// TIA Portal V20 export
// export: Created 2025-12-01T14:56:43.4302356Z, ExportSetting None, DisplayName Totally Integrated Automation Portal, DisplayVersion V20 Update 3, DisplayName TIA Portal Openness, DisplayVersion V20 Update 3, DisplayName TIA Portal Version Control Interface, DisplayVersion V20 Update 3, DisplayName STEP 7 Professional, DisplayVersion V20 Update 3, DisplayName STEP 7 Safety, DisplayVersion V20 Update 2, DisplayName WinCC Basic/Comfort/Advanced, DisplayVersion V20 Update 3, DisplayName WinCC Professional, DisplayVersion V20 Update 3, DisplayName WinCC Unified, DisplayVersion V20 Update 3
FUNCTION_BLOCK "FB243_M_STV_Carga_E1_S3_Doble"   // FB243, LAD
TITLE = Control del Ramal de Salidas
{ S7_Optimized_Access := 'FALSE' }
AUTHOR : VTD
NAME : 20160509
VERSION : 3.5
// stored: AutoNumber false, SetENOAutomatically false
   VAR_INPUT
      Mesa : UInt;   // Mesa de la FB
      Error_Tx : Bool;   // Error en el Tx
      EnTension : Bool;   // Existe Tension en la Mesa
      Termico_Tx : Bool;   // Proteccion del Tx
      pHsMx_1 : Bool;   // pHs de la Mesa
      pHsMx_2 : Bool;   // pHs de la Mesa
      pHsMx_PR1 : Bool;   // pHs de Protrusion de la Mesa. Nota: No existe >> ON
      pHsMx_PR3 : Bool;   // pHs de Protrusion de la Mesa. Nota: No existe >> ON
      Avance_Tx : Bool;   // Avance del Tx
      LoadArrival : Bool;   // Load Arrival >>> VTD
      LoadComplete : Bool;   // LoadComplete >>> VTD
      MAnt_DescargaAct : Bool;   // E1 >> Mesa Anterior DescargaAct
      AVTF_MAnt_Mx : Bool;   // E1 >> Mesa Anterior AVTF
      P_Mens_MAnt_Mx : Bool;   // E1 >> Mesa Anterior P_Mens
      MAnt_CargaLarga : Bool;   // E1 >> Mesa Anterior Carga Larga
      Mx_VelocidadLenta_In : Bool;   // Forzar a Velociada Lenta
      F_EnvMens_Mx : Bool;   // Fin de Envio de Mensaje
      OrdSal_S00 : Bool;   // Orden de Salida hacia el VTD
      V_CNT_pHsMx : Int := 1000;   // Valor de Presencia
      V_CNT_pHsMx_FTF : Int := 200;   // Valor para activar FTF. Nota: < = V_CNT_pHsMx.
      V_CNTSeg_pHsMx : Int := 2000;   // Valor de Seguriadad para Presencia
      V_CNT_PasoLenta : Int := 2000;   // Valor de Paso a Lenta
      V_CNT_ApHsMx : Int := 200;   // Valor de Ausencia
      V_CNTSeg_ApHsMx : Int := 2000;   // Valor de Seguriadad para Ausencia
      V_TOut_Tx_Mx : Int := 15000;   // TimeOut de Entrada por E1
      V_TOut_Interlock : Int := 5000;   // TimeOut de Fin del Interlock con el VTD
      V_TMP_Protrusion : Int := 200;   // TMP de Protrusion
      V_CNT_PerdidapHs : Int := 1000;   // CNT de Perdida de pHs
   END_VAR
   VAR_OUTPUT
      P_EnvMens_PMx : Bool;   // Permiso de Enviar Mensaje de Presencia
      P_EnvMens_AMx : Bool;   // Permiso de Enviar Mensaje de Ausencia
      P_RecepOK_Mx : Bool;   // Recepcion OK
      PTF_MAnt_Mx : Bool;   // E1 >> Mesa Anterior PTF
      FTF_MAnt_Mx : Bool;   // E1 >> Mesa Anterior FTF
   END_VAR
   VAR
      Anular_prE1 : Bool;   // ???
      Anular_prS3 : Bool;   // ???
      Mx_ET00 : Bool;
      Mx_ET01 : Bool;
      Mx_ET02 : Bool;
      Mx_ET06 : Bool;
      Mx_ET07 : Bool;
      Mx_ET08 : Bool;
      Mx_ET09 : Bool;
      Mx_ET10 : Bool;
      Mx_ET10Doble : Bool;
      Mx_ET11 : Bool;
      Mx_ET12 : Bool;
      Mx_ET110 : Bool;
      Mx_ET111 : Bool;
      Mx_ET50 : Bool;
      Mx_ET51 : Bool;
      Mx_ET52 : Bool;
      Mx_ET150 : Bool;
      Mx_ET151 : Bool;
      Mx_ET152 : Bool;
      MemoriaCargaDoble : Bool;   // Interna >>> Memoria Carga Doble
      ProtocoloIniciado : Bool;   // Iniciado el Envio del Mensaje de Presencia
      CNT_pHsMx_FTF_OK : Bool;   // Enviar ya FTF
      STAT_EnvMens_PMx : Bool;   // Interna >> Envio del Mensaje de Presencia
      STAT_EnvMens_AMx : Bool;   // Interna >> Envio de Mensaje de Ausencia
      STAT_FTF_MAnt_Mx : Bool;   // Interna >> FTF de MAnt >> Mx
      CNT_pHsMx { S7_SetPoint := 'True'} : "FB910_CNT_UHS";   // CNT de la Presencia
      CNTSeg_pHsMx { S7_SetPoint := 'True'} : "FB910_CNT_UHS";   // CNT de Seguridad de la Presencia
      CNT_ApHsMx { S7_SetPoint := 'True'} : "FB910_CNT_UHS";   // CNT de la Ausencia
      CNTSeg_ApHsMx { S7_SetPoint := 'True'} : "FB910_CNT_UHS";   // CNT de Seguridad de la Ausencia
      TMP_EnTension { S7_SetPoint := 'True'} : "FB910_CNT_UHS";
      TOut_Av_Mx { S7_SetPoint := 'True'} : "FB910_CNT_UHS";   // Time Out de Entrada de E1
      TOut_Interlock { S7_SetPoint := 'True'} : "FB910_CNT_UHS";   // Time Out de Fin de Interlock con el VTD
      TMP_Protrusion { S7_SetPoint := 'True'} : "FB910_CNT_UHS";   // TMP de la Protrusion
      Interlock_manual { S7_SetPoint := 'True'} : "UDT_Interlock_manual_STV";
      CNT_PerdidapHs { S7_SetPoint := 'True'} : "FB910_CNT_UHS";   // CNT de Perdida de pHs
   END_VAR
   VAR_TEMP
      EstadoZona : "EstadoZona";   // Estado de Zona de la Mesa
      EstadoVI : "EstadosMesa";   // Estado del Vehiculo Inteliguente de la Mesa
      ConfigFB : "UDT_ConfigFB";   // Configuracion de la FB de la Mesa
      Interlock : "UDT_Interlock_STV";
      V_Protrusion : Int;
      retval : Int;
      cero : USInt;
      Aux_ET00 : Bool;
   END_VAR
BEGIN

REGION Network 1: INICIALIZAR - Recoger las Variables de Estado de la Mesa
   // Se recoge - Estado_CBx
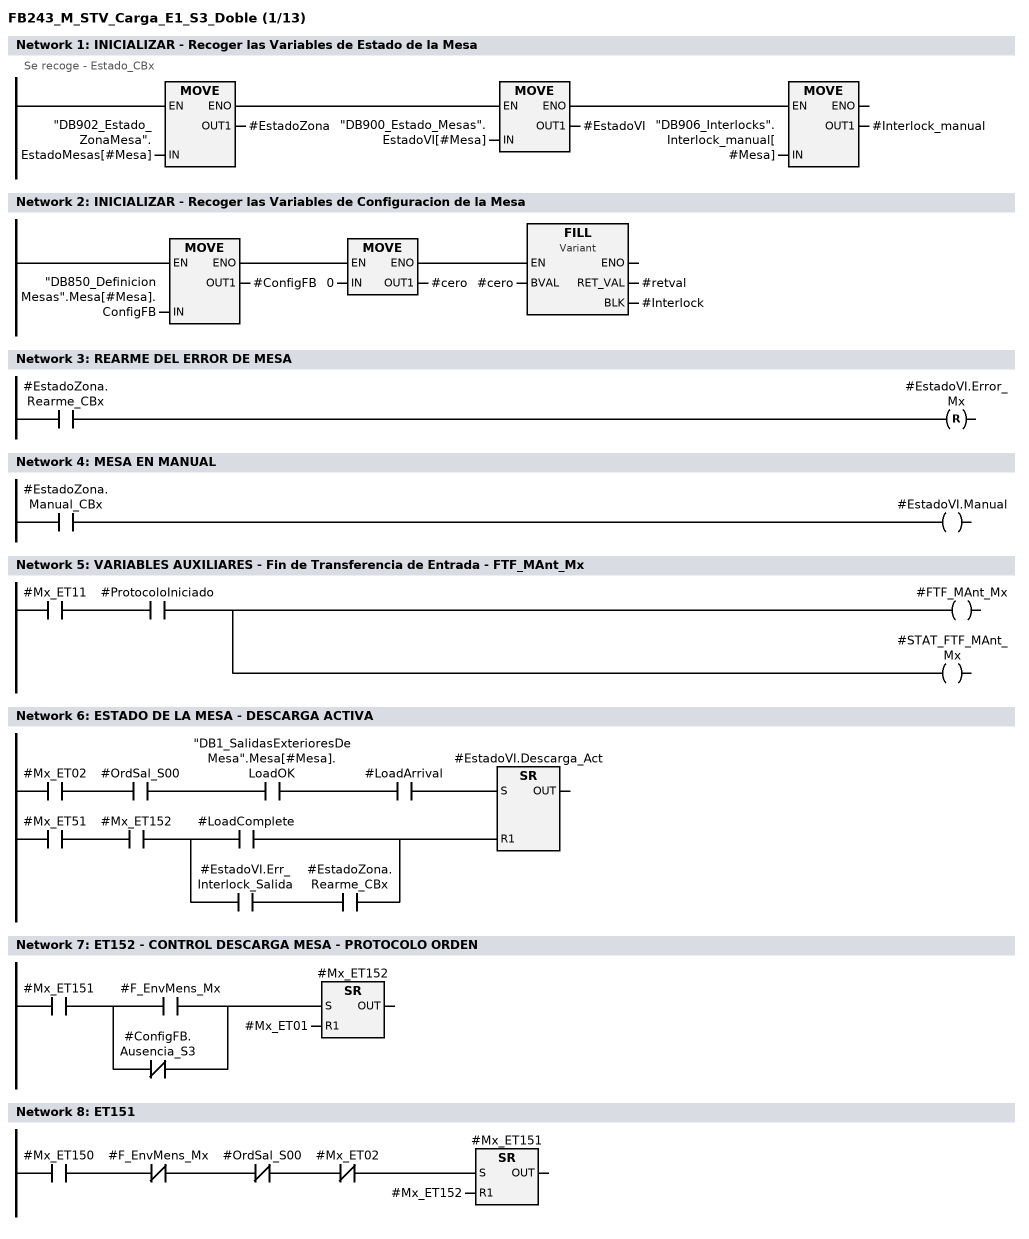
   RUNG wire#powerrail
      Move(in := "DB902_Estado_ZonaMesa".EstadoMesas[#Mesa], out1 => #EstadoZona)
      Move(in := "DB900_Estado_Mesas".EstadoVI[#Mesa], out1 => #EstadoVI)
      Move(in := "DB906_Interlocks".Interlock_manual[#Mesa], out1 => #Interlock_manual)
   END_RUNG
   // the same network as SCL:
   #EstadoZona := "DB902_Estado_ZonaMesa".EstadoMesas[#Mesa];
   #EstadoVI := "DB900_Estado_Mesas".EstadoVI[#Mesa];
   #Interlock_manual := "DB906_Interlocks".Interlock_manual[#Mesa];
END_REGION

REGION Network 2: INICIALIZAR - Recoger las Variables de Configuracion de la Mesa
   RUNG wire#powerrail
      Move(in := "DB850_DefinicionMesas".Mesa[#Mesa].ConfigFB, out1 => #ConfigFB)
      Move(in := 0, out1 => #cero)
      { S7_Templates := "ptr_type := Variant" } FILL(BVAL := #cero, RET_VAL => #retval, BLK => #Interlock)
   END_RUNG
   // the same network as SCL:
   #ConfigFB := "DB850_DefinicionMesas".Mesa[#Mesa].ConfigFB;
   #cero := 0;
   #retval := FILL(BVAL := #cero, BLK => #Interlock);
END_REGION

REGION Network 3: REARME DEL ERROR DE MESA
   RUNG wire#powerrail
      Contact( #EstadoZona.Rearme_CBx )
      R_Coil( #EstadoVI.Error_Mx )
   END_RUNG
   // the same network as SCL:
   IF #EstadoZona.Rearme_CBx THEN #EstadoVI.Error_Mx := FALSE; END_IF;
END_REGION

REGION Network 4: MESA EN MANUAL
   RUNG wire#powerrail
      Contact( #EstadoZona.Manual_CBx )
      Coil( #EstadoVI.Manual )
   END_RUNG
   // the same network as SCL:
   #EstadoVI.Manual := #EstadoZona.Manual_CBx;
END_REGION

REGION Network 5: VARIABLES AUXILIARES - Fin de Transferencia de Entrada - FTF_MAnt_Mx
   RUNG wire#powerrail
      Contact( #Mx_ET11 )
      Contact( #ProtocoloIniciado )
      wire#w1
      Coil( #FTF_MAnt_Mx )
   END_RUNG
   RUNG wire#w1
      Coil( #STAT_FTF_MAnt_Mx )
   END_RUNG
   // the same network as SCL:
   #FTF_MAnt_Mx := #Mx_ET11 AND #ProtocoloIniciado;
   #STAT_FTF_MAnt_Mx := #FTF_MAnt_Mx;
END_REGION

REGION Network 6: ESTADO DE LA MESA - DESCARGA ACTIVA
   RUNG wire#powerrail
      Contact( #Mx_ET02 )
      Contact( #OrdSal_S00 )
      Contact( "DB1_SalidasExterioresDeMesa".Mesa[#Mesa].LoadOK )
      Contact( #LoadArrival )
      S_SR(operand := #EstadoVI.Descarga_Act, r1 := wire#w2)
   END_RUNG
   RUNG wire#powerrail
      Contact( #Mx_ET51 )
      Contact( #Mx_ET152 )
      wire#w1
      Contact( #LoadComplete )
   END_RUNG wire#w2
   RUNG wire#w1
      Contact( #EstadoVI.Err_Interlock_Salida )
      Contact( #EstadoZona.Rearme_CBx )
   END_RUNG wire#w2
   // the same network as SCL:
   IF #Mx_ET02 AND #OrdSal_S00 AND "DB1_SalidasExterioresDeMesa".Mesa[#Mesa].LoadOK AND #LoadArrival THEN
       #EstadoVI.Descarga_Act := TRUE;   // SR flip-flop
   END_IF;
   IF #Mx_ET51 AND #Mx_ET152 AND (#LoadComplete OR (#EstadoVI.Err_Interlock_Salida AND #EstadoZona.Rearme_CBx)) THEN
       #EstadoVI.Descarga_Act := FALSE;
   END_IF;
END_REGION

REGION Network 7: ET152 - CONTROL DESCARGA MESA - PROTOCOLO ORDEN
   RUNG wire#powerrail
      Contact( #Mx_ET151 )
      wire#w1
      Contact( #F_EnvMens_Mx )
      wire#w2
      S_SR(operand := #Mx_ET152, r1 := #Mx_ET01)
   END_RUNG
   RUNG wire#w1
      I_Contact( #ConfigFB.Ausencia_S3 )
   END_RUNG wire#w2
   // the same network as SCL:
   IF #Mx_ET151 AND (#F_EnvMens_Mx OR NOT #ConfigFB.Ausencia_S3) THEN
       #Mx_ET152 := TRUE;   // SR flip-flop
   END_IF;
   IF #Mx_ET01 THEN #Mx_ET152 := FALSE; END_IF;
END_REGION

REGION Network 8: ET151
   RUNG wire#powerrail
      Contact( #Mx_ET150 )
      I_Contact( #F_EnvMens_Mx )
      I_Contact( #OrdSal_S00 )
      I_Contact( #Mx_ET02 )
      S_SR(operand := #Mx_ET151, r1 := #Mx_ET152)
   END_RUNG
   // the same network as SCL:
   IF #Mx_ET150 AND NOT #F_EnvMens_Mx AND NOT #OrdSal_S00 AND NOT #Mx_ET02 THEN
       #Mx_ET151 := TRUE;   // SR flip-flop
   END_IF;
   IF #Mx_ET152 THEN #Mx_ET151 := FALSE; END_IF;
END_REGION

REGION Network 9: ET150
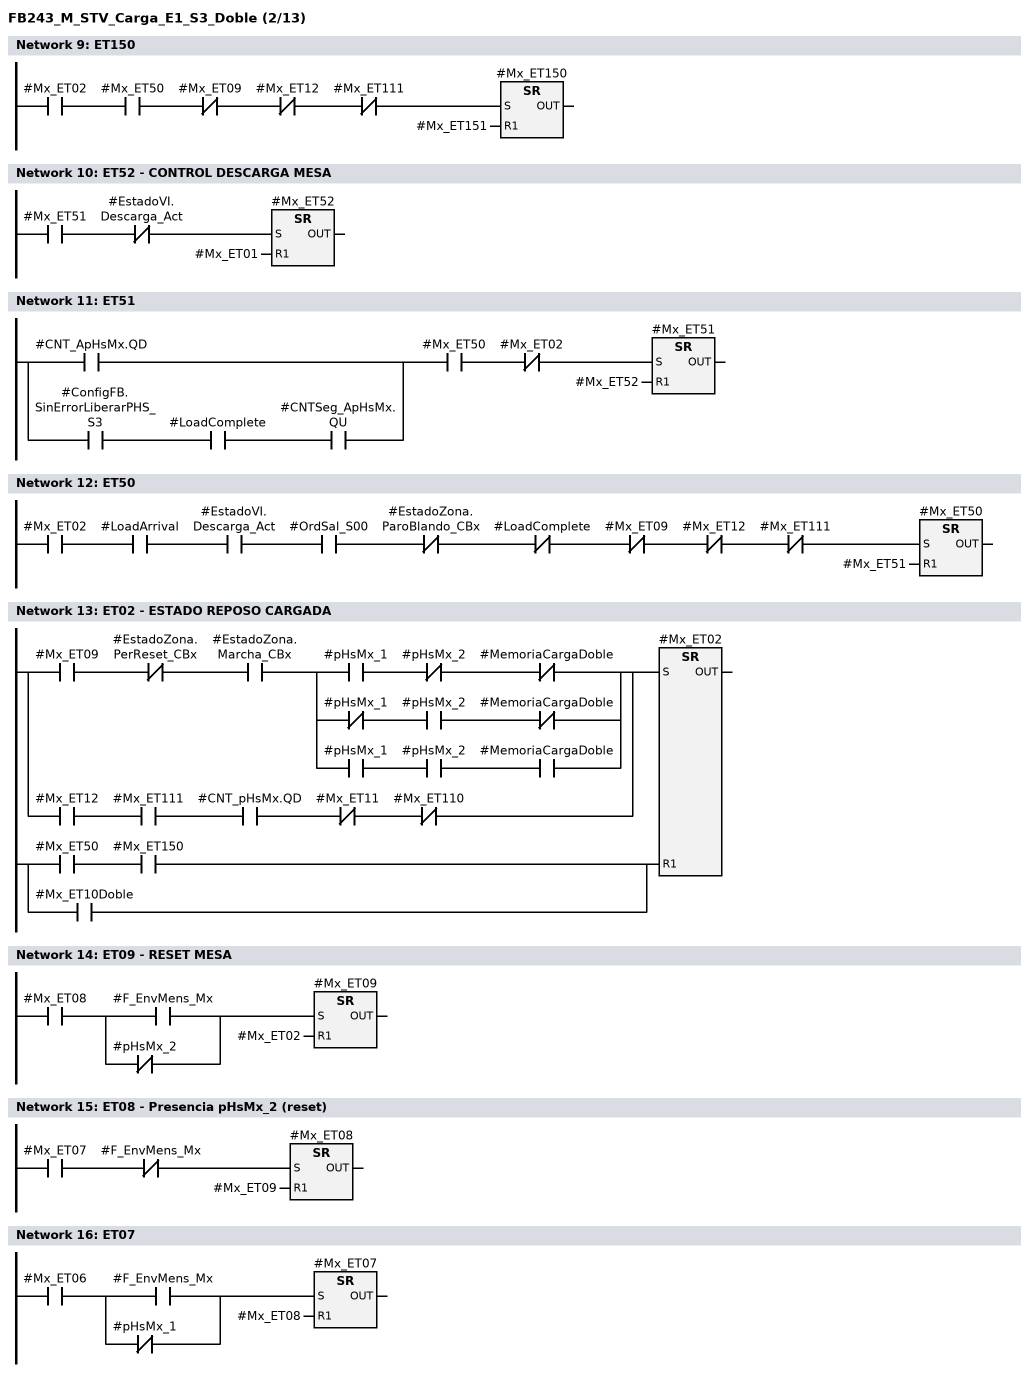
   RUNG wire#powerrail
      Contact( #Mx_ET02 )
      Contact( #Mx_ET50 )
      I_Contact( #Mx_ET09 )
      I_Contact( #Mx_ET12 )
      I_Contact( #Mx_ET111 )
      S_SR(operand := #Mx_ET150, r1 := #Mx_ET151)
   END_RUNG
   // the same network as SCL:
   IF #Mx_ET02 AND #Mx_ET50 AND NOT #Mx_ET09 AND NOT #Mx_ET12 AND NOT #Mx_ET111 THEN
       #Mx_ET150 := TRUE;   // SR flip-flop
   END_IF;
   IF #Mx_ET151 THEN #Mx_ET150 := FALSE; END_IF;
END_REGION

REGION Network 10: ET52 - CONTROL DESCARGA MESA
   RUNG wire#powerrail
      Contact( #Mx_ET51 )
      I_Contact( #EstadoVI.Descarga_Act )
      S_SR(operand := #Mx_ET52, r1 := #Mx_ET01)
   END_RUNG
   // the same network as SCL:
   IF #Mx_ET51 AND NOT #EstadoVI.Descarga_Act THEN
       #Mx_ET52 := TRUE;   // SR flip-flop
   END_IF;
   IF #Mx_ET01 THEN #Mx_ET52 := FALSE; END_IF;
END_REGION

REGION Network 11: ET51
   RUNG wire#powerrail
      Contact( #CNT_ApHsMx.QD )
      wire#w1
      Contact( #Mx_ET50 )
      I_Contact( #Mx_ET02 )
      S_SR(operand := #Mx_ET51, r1 := #Mx_ET52)
   END_RUNG
   RUNG wire#powerrail
      Contact( #ConfigFB.SinErrorLiberarPHS_S3 )
      Contact( #LoadComplete )
      Contact( #CNTSeg_ApHsMx.QU )
   END_RUNG wire#w1
   // the same network as SCL:
   IF (#CNT_ApHsMx.QD OR (#ConfigFB.SinErrorLiberarPHS_S3 AND #LoadComplete AND #CNTSeg_ApHsMx.QU)) AND #Mx_ET50 AND NOT #Mx_ET02 THEN
       #Mx_ET51 := TRUE;   // SR flip-flop
   END_IF;
   IF #Mx_ET52 THEN #Mx_ET51 := FALSE; END_IF;
END_REGION

REGION Network 12: ET50
   RUNG wire#powerrail
      Contact( #Mx_ET02 )
      Contact( #LoadArrival )
      Contact( #EstadoVI.Descarga_Act )
      Contact( #OrdSal_S00 )
      I_Contact( #EstadoZona.ParoBlando_CBx )
      I_Contact( #LoadComplete )
      I_Contact( #Mx_ET09 )
      I_Contact( #Mx_ET12 )
      I_Contact( #Mx_ET111 )
      S_SR(operand := #Mx_ET50, r1 := #Mx_ET51)
   END_RUNG
   // the same network as SCL:
   IF #Mx_ET02 AND #LoadArrival AND #EstadoVI.Descarga_Act AND #OrdSal_S00 AND NOT #EstadoZona.ParoBlando_CBx AND NOT #LoadComplete AND NOT #Mx_ET09 AND NOT #Mx_ET12 AND NOT #Mx_ET111 THEN
       #Mx_ET50 := TRUE;   // SR flip-flop
   END_IF;
   IF #Mx_ET51 THEN #Mx_ET50 := FALSE; END_IF;
END_REGION

REGION Network 13: ET02 - ESTADO REPOSO CARGADA
   RUNG wire#powerrail
      Contact( #Mx_ET09 )
      I_Contact( #EstadoZona.PerReset_CBx )
      Contact( #EstadoZona.Marcha_CBx )
      wire#w1
      Contact( #pHsMx_1 )
      I_Contact( #pHsMx_2 )
      I_Contact( #MemoriaCargaDoble )
      wire#w2
      S_SR(operand := #Mx_ET02, r1 := wire#w3)
   END_RUNG
   RUNG wire#w1
      I_Contact( #pHsMx_1 )
      Contact( #pHsMx_2 )
      I_Contact( #MemoriaCargaDoble )
   END_RUNG wire#w2
   RUNG wire#w1
      Contact( #pHsMx_1 )
      Contact( #pHsMx_2 )
      Contact( #MemoriaCargaDoble )
   END_RUNG wire#w2
   RUNG wire#powerrail
      Contact( #Mx_ET12 )
      Contact( #Mx_ET111 )
      Contact( #CNT_pHsMx.QD )
      I_Contact( #Mx_ET11 )
      I_Contact( #Mx_ET110 )
   END_RUNG wire#w2
   RUNG wire#powerrail
      Contact( #Mx_ET50 )
      Contact( #Mx_ET150 )
   END_RUNG wire#w3
   RUNG wire#powerrail
      Contact( #Mx_ET10Doble )
   END_RUNG wire#w3
   // the same network as SCL:
   IF (#Mx_ET09 AND NOT #EstadoZona.PerReset_CBx AND #EstadoZona.Marcha_CBx AND ((#pHsMx_1 AND NOT #pHsMx_2 AND NOT #MemoriaCargaDoble) OR (NOT #pHsMx_1 AND #pHsMx_2 AND NOT #MemoriaCargaDoble) OR (#pHsMx_1 AND #pHsMx_2 AND #MemoriaCargaDoble))) OR (#Mx_ET12 AND #Mx_ET111 AND #CNT_pHsMx.QD AND NOT #Mx_ET11 AND NOT #Mx_ET110) THEN
       #Mx_ET02 := TRUE;   // SR flip-flop
   END_IF;
   IF (#Mx_ET50 AND #Mx_ET150) OR #Mx_ET10Doble THEN #Mx_ET02 := FALSE; END_IF;
END_REGION

REGION Network 14: ET09 - RESET MESA
   RUNG wire#powerrail
      Contact( #Mx_ET08 )
      wire#w1
      Contact( #F_EnvMens_Mx )
      wire#w2
      S_SR(operand := #Mx_ET09, r1 := #Mx_ET02)
   END_RUNG
   RUNG wire#w1
      I_Contact( #pHsMx_2 )
   END_RUNG wire#w2
   // the same network as SCL:
   IF #Mx_ET08 AND (#F_EnvMens_Mx OR NOT #pHsMx_2) THEN
       #Mx_ET09 := TRUE;   // SR flip-flop
   END_IF;
   IF #Mx_ET02 THEN #Mx_ET09 := FALSE; END_IF;
END_REGION

REGION Network 15: ET08 - Presencia pHsMx_2 (reset)
   RUNG wire#powerrail
      Contact( #Mx_ET07 )
      I_Contact( #F_EnvMens_Mx )
      S_SR(operand := #Mx_ET08, r1 := #Mx_ET09)
   END_RUNG
   // the same network as SCL:
   IF #Mx_ET07 AND NOT #F_EnvMens_Mx THEN
       #Mx_ET08 := TRUE;   // SR flip-flop
   END_IF;
   IF #Mx_ET09 THEN #Mx_ET08 := FALSE; END_IF;
END_REGION

REGION Network 16: ET07
   RUNG wire#powerrail
      Contact( #Mx_ET06 )
      wire#w1
      Contact( #F_EnvMens_Mx )
      wire#w2
      S_SR(operand := #Mx_ET07, r1 := #Mx_ET08)
   END_RUNG
   RUNG wire#w1
      I_Contact( #pHsMx_1 )
   END_RUNG wire#w2
   // the same network as SCL:
   IF #Mx_ET06 AND (#F_EnvMens_Mx OR NOT #pHsMx_1) THEN
       #Mx_ET07 := TRUE;   // SR flip-flop
   END_IF;
   IF #Mx_ET08 THEN #Mx_ET07 := FALSE; END_IF;
END_REGION

REGION Network 17: ET06 - Presencia pHsMx_1 (reset)
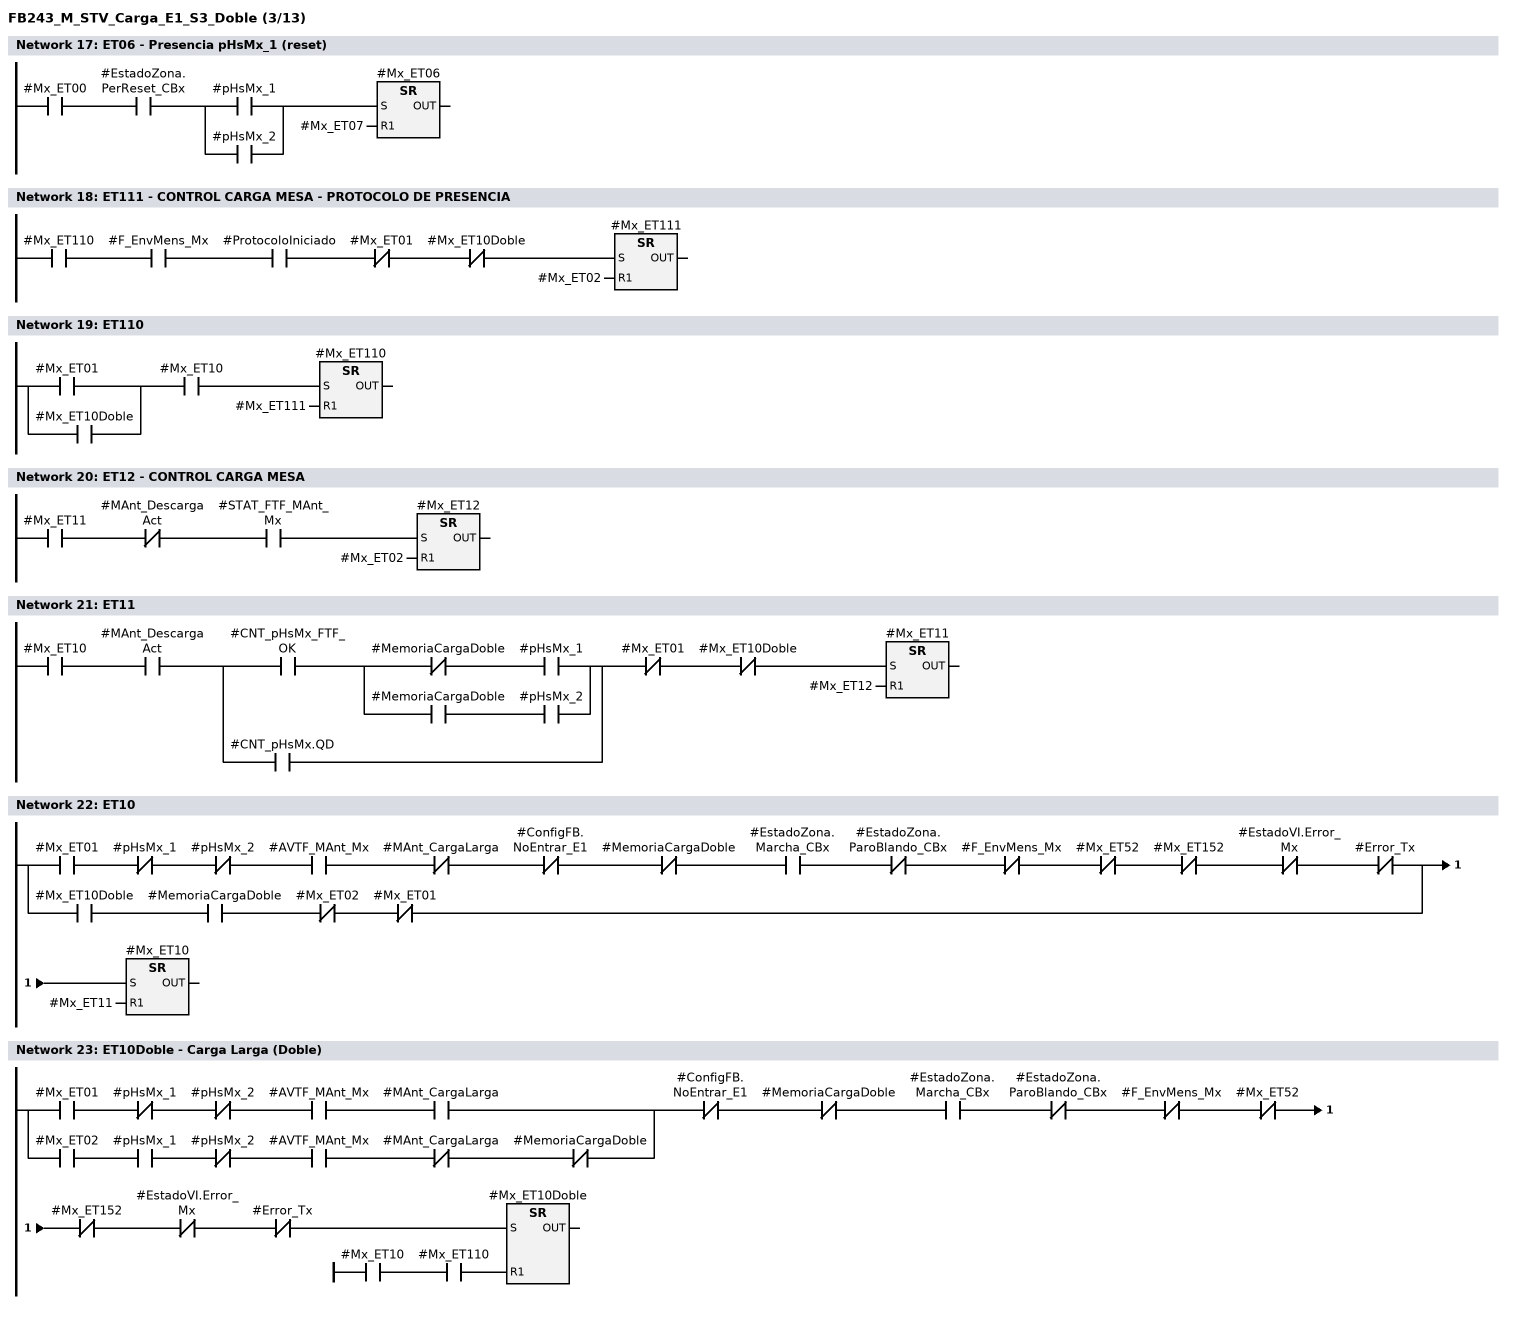
   RUNG wire#powerrail
      Contact( #Mx_ET00 )
      Contact( #EstadoZona.PerReset_CBx )
      wire#w1
      Contact( #pHsMx_1 )
      wire#w2
      S_SR(operand := #Mx_ET06, r1 := #Mx_ET07)
   END_RUNG
   RUNG wire#w1
      Contact( #pHsMx_2 )
   END_RUNG wire#w2
   // the same network as SCL:
   IF #Mx_ET00 AND #EstadoZona.PerReset_CBx AND (#pHsMx_1 OR #pHsMx_2) THEN
       #Mx_ET06 := TRUE;   // SR flip-flop
   END_IF;
   IF #Mx_ET07 THEN #Mx_ET06 := FALSE; END_IF;
END_REGION

REGION Network 18: ET111 - CONTROL CARGA MESA - PROTOCOLO DE PRESENCIA
   RUNG wire#powerrail
      Contact( #Mx_ET110 )
      Contact( #F_EnvMens_Mx )
      Contact( #ProtocoloIniciado )
      I_Contact( #Mx_ET01 )
      I_Contact( #Mx_ET10Doble )
      S_SR(operand := #Mx_ET111, r1 := #Mx_ET02)
   END_RUNG
   // the same network as SCL:
   IF #Mx_ET110 AND #F_EnvMens_Mx AND #ProtocoloIniciado AND NOT #Mx_ET01 AND NOT #Mx_ET10Doble THEN
       #Mx_ET111 := TRUE;   // SR flip-flop
   END_IF;
   IF #Mx_ET02 THEN #Mx_ET111 := FALSE; END_IF;
END_REGION

REGION Network 19: ET110
   RUNG wire#powerrail
      Contact( #Mx_ET01 )
      wire#w1
      Contact( #Mx_ET10 )
      S_SR(operand := #Mx_ET110, r1 := #Mx_ET111)
   END_RUNG
   RUNG wire#powerrail
      Contact( #Mx_ET10Doble )
   END_RUNG wire#w1
   // the same network as SCL:
   IF (#Mx_ET01 OR #Mx_ET10Doble) AND #Mx_ET10 THEN
       #Mx_ET110 := TRUE;   // SR flip-flop
   END_IF;
   IF #Mx_ET111 THEN #Mx_ET110 := FALSE; END_IF;
END_REGION

REGION Network 20: ET12 - CONTROL CARGA MESA
   RUNG wire#powerrail
      Contact( #Mx_ET11 )
      I_Contact( #MAnt_DescargaAct )
      Contact( #STAT_FTF_MAnt_Mx )
      S_SR(operand := #Mx_ET12, r1 := #Mx_ET02)
   END_RUNG
   // the same network as SCL:
   IF #Mx_ET11 AND NOT #MAnt_DescargaAct AND #STAT_FTF_MAnt_Mx THEN
       #Mx_ET12 := TRUE;   // SR flip-flop
   END_IF;
   IF #Mx_ET02 THEN #Mx_ET12 := FALSE; END_IF;
END_REGION

REGION Network 21: ET11
   RUNG wire#powerrail
      Contact( #Mx_ET10 )
      Contact( #MAnt_DescargaAct )
      wire#w1
      Contact( #CNT_pHsMx_FTF_OK )
      wire#w2
      I_Contact( #MemoriaCargaDoble )
      Contact( #pHsMx_1 )
      wire#w3
      I_Contact( #Mx_ET01 )
      I_Contact( #Mx_ET10Doble )
      S_SR(operand := #Mx_ET11, r1 := #Mx_ET12)
   END_RUNG
   RUNG wire#w2
      Contact( #MemoriaCargaDoble )
      Contact( #pHsMx_2 )
   END_RUNG wire#w3
   RUNG wire#w1
      Contact( #CNT_pHsMx.QD )
   END_RUNG wire#w3
   // the same network as SCL:
   IF #Mx_ET10 AND #MAnt_DescargaAct AND ((#CNT_pHsMx_FTF_OK AND ((NOT #MemoriaCargaDoble AND #pHsMx_1) OR (#MemoriaCargaDoble AND #pHsMx_2))) OR #CNT_pHsMx.QD) AND NOT #Mx_ET01 AND NOT #Mx_ET10Doble THEN
       #Mx_ET11 := TRUE;   // SR flip-flop
   END_IF;
   IF #Mx_ET12 THEN #Mx_ET11 := FALSE; END_IF;
END_REGION

REGION Network 22: ET10
   RUNG wire#powerrail
      Contact( #Mx_ET01 )
      I_Contact( #pHsMx_1 )
      I_Contact( #pHsMx_2 )
      Contact( #AVTF_MAnt_Mx )
      I_Contact( #MAnt_CargaLarga )
      I_Contact( #ConfigFB.NoEntrar_E1 )
      I_Contact( #MemoriaCargaDoble )
      Contact( #EstadoZona.Marcha_CBx )
      I_Contact( #EstadoZona.ParoBlando_CBx )
      I_Contact( #F_EnvMens_Mx )
      I_Contact( #Mx_ET52 )
      I_Contact( #Mx_ET152 )
      I_Contact( #EstadoVI.Error_Mx )
      I_Contact( #Error_Tx )
      wire#w1
      S_SR(operand := #Mx_ET10, r1 := #Mx_ET11)
   END_RUNG
   RUNG wire#powerrail
      Contact( #Mx_ET10Doble )
      Contact( #MemoriaCargaDoble )
      I_Contact( #Mx_ET02 )
      I_Contact( #Mx_ET01 )
   END_RUNG wire#w1
   // the same network as SCL:
   IF (#Mx_ET01 AND NOT #pHsMx_1 AND NOT #pHsMx_2 AND #AVTF_MAnt_Mx AND NOT #MAnt_CargaLarga AND NOT #ConfigFB.NoEntrar_E1 AND NOT #MemoriaCargaDoble AND #EstadoZona.Marcha_CBx AND NOT #EstadoZona.ParoBlando_CBx AND NOT #F_EnvMens_Mx AND NOT #Mx_ET52 AND NOT #Mx_ET152 AND NOT #EstadoVI.Error_Mx AND NOT #Error_Tx) OR (#Mx_ET10Doble AND #MemoriaCargaDoble AND NOT #Mx_ET02 AND NOT #Mx_ET01) THEN
       #Mx_ET10 := TRUE;   // SR flip-flop
   END_IF;
   IF #Mx_ET11 THEN #Mx_ET10 := FALSE; END_IF;
END_REGION

REGION Network 23: ET10Doble - Carga Larga (Doble)
   RUNG wire#powerrail
      Contact( #Mx_ET01 )
      I_Contact( #pHsMx_1 )
      I_Contact( #pHsMx_2 )
      Contact( #AVTF_MAnt_Mx )
      Contact( #MAnt_CargaLarga )
      wire#w1
      I_Contact( #ConfigFB.NoEntrar_E1 )
      I_Contact( #MemoriaCargaDoble )
      Contact( #EstadoZona.Marcha_CBx )
      I_Contact( #EstadoZona.ParoBlando_CBx )
      I_Contact( #F_EnvMens_Mx )
      I_Contact( #Mx_ET52 )
      I_Contact( #Mx_ET152 )
      I_Contact( #EstadoVI.Error_Mx )
      I_Contact( #Error_Tx )
      S_SR(operand := #Mx_ET10Doble, r1 := wire#w2)
   END_RUNG
   RUNG wire#powerrail
      Contact( #Mx_ET02 )
      Contact( #pHsMx_1 )
      I_Contact( #pHsMx_2 )
      Contact( #AVTF_MAnt_Mx )
      I_Contact( #MAnt_CargaLarga )
      I_Contact( #MemoriaCargaDoble )
   END_RUNG wire#w1
   RUNG wire#powerrail
      Contact( #Mx_ET10 )
      Contact( #Mx_ET110 )
   END_RUNG wire#w2
   // the same network as SCL:
   IF ((#Mx_ET01 AND NOT #pHsMx_1 AND NOT #pHsMx_2 AND #AVTF_MAnt_Mx AND #MAnt_CargaLarga) OR (#Mx_ET02 AND #pHsMx_1 AND NOT #pHsMx_2 AND #AVTF_MAnt_Mx AND NOT #MAnt_CargaLarga AND NOT #MemoriaCargaDoble)) AND NOT #ConfigFB.NoEntrar_E1 AND NOT #MemoriaCargaDoble AND #EstadoZona.Marcha_CBx AND NOT #EstadoZona.ParoBlando_CBx AND NOT #F_EnvMens_Mx AND NOT #Mx_ET52 AND NOT #Mx_ET152 AND NOT #EstadoVI.Error_Mx AND NOT #Error_Tx THEN
       #Mx_ET10Doble := TRUE;   // SR flip-flop
   END_IF;
   IF #Mx_ET10 AND #Mx_ET110 THEN #Mx_ET10Doble := FALSE; END_IF;
END_REGION

REGION Network 24: ET01 - ESTADO REPOSO VACIO
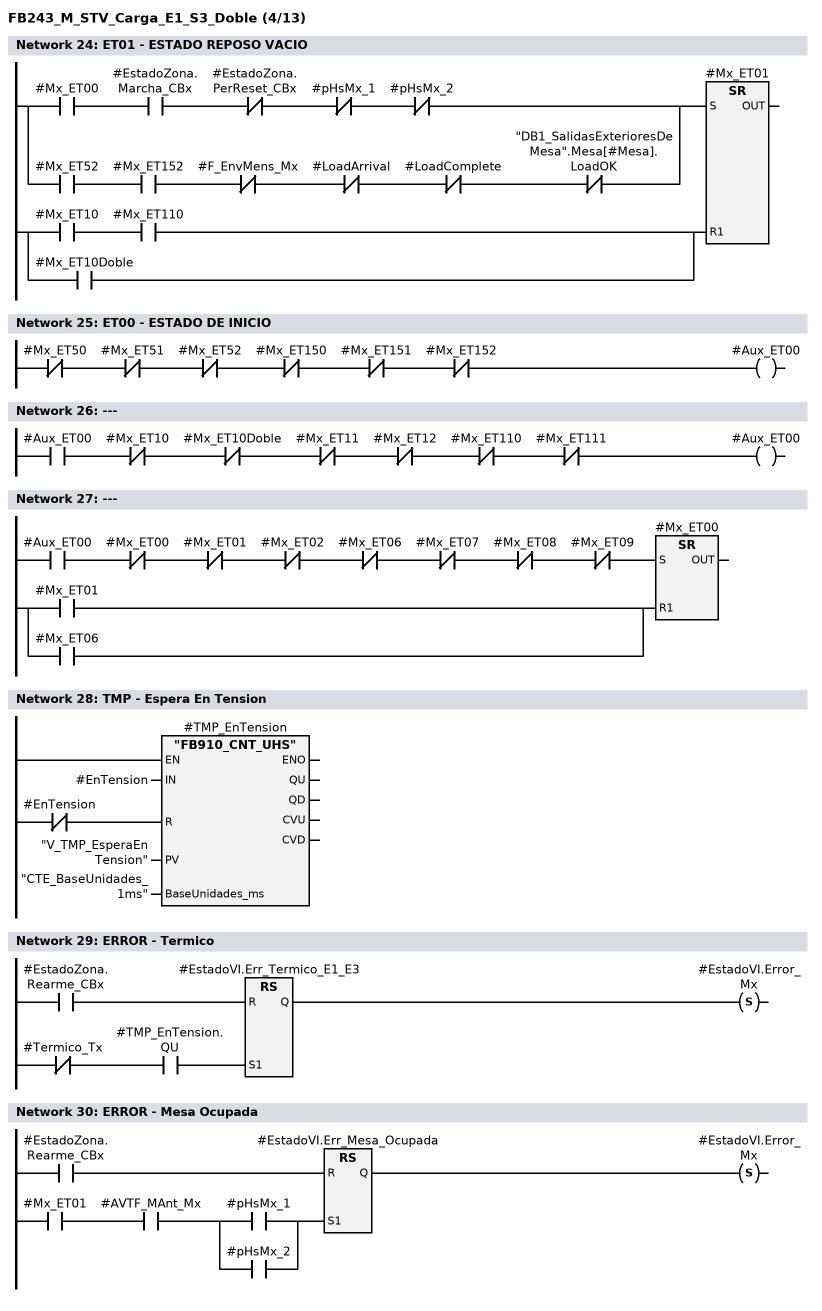
   RUNG wire#powerrail
      Contact( #Mx_ET00 )
      Contact( #EstadoZona.Marcha_CBx )
      I_Contact( #EstadoZona.PerReset_CBx )
      I_Contact( #pHsMx_1 )
      I_Contact( #pHsMx_2 )
      wire#w1
      S_SR(operand := #Mx_ET01, r1 := wire#w2)
   END_RUNG
   RUNG wire#powerrail
      Contact( #Mx_ET52 )
      Contact( #Mx_ET152 )
      I_Contact( #F_EnvMens_Mx )
      I_Contact( #LoadArrival )
      I_Contact( #LoadComplete )
      I_Contact( "DB1_SalidasExterioresDeMesa".Mesa[#Mesa].LoadOK )
   END_RUNG wire#w1
   RUNG wire#powerrail
      Contact( #Mx_ET10 )
      Contact( #Mx_ET110 )
   END_RUNG wire#w2
   RUNG wire#powerrail
      Contact( #Mx_ET10Doble )
   END_RUNG wire#w2
   // the same network as SCL:
   IF (#Mx_ET00 AND #EstadoZona.Marcha_CBx AND NOT #EstadoZona.PerReset_CBx AND NOT #pHsMx_1 AND NOT #pHsMx_2) OR (#Mx_ET52 AND #Mx_ET152 AND NOT #F_EnvMens_Mx AND NOT #LoadArrival AND NOT #LoadComplete AND NOT "DB1_SalidasExterioresDeMesa".Mesa[#Mesa].LoadOK) THEN
       #Mx_ET01 := TRUE;   // SR flip-flop
   END_IF;
   IF (#Mx_ET10 AND #Mx_ET110) OR #Mx_ET10Doble THEN #Mx_ET01 := FALSE; END_IF;
END_REGION

REGION Network 25: ET00 - ESTADO DE INICIO
   RUNG wire#powerrail
      I_Contact( #Mx_ET50 )
      I_Contact( #Mx_ET51 )
      I_Contact( #Mx_ET52 )
      I_Contact( #Mx_ET150 )
      I_Contact( #Mx_ET151 )
      I_Contact( #Mx_ET152 )
      Coil( #Aux_ET00 )
   END_RUNG
   // the same network as SCL:
   #Aux_ET00 := NOT #Mx_ET50 AND NOT #Mx_ET51 AND NOT #Mx_ET52 AND NOT #Mx_ET150 AND NOT #Mx_ET151 AND NOT #Mx_ET152;
END_REGION

REGION Network 26: ---
   RUNG wire#powerrail
      Contact( #Aux_ET00 )
      I_Contact( #Mx_ET10 )
      I_Contact( #Mx_ET10Doble )
      I_Contact( #Mx_ET11 )
      I_Contact( #Mx_ET12 )
      I_Contact( #Mx_ET110 )
      I_Contact( #Mx_ET111 )
      Coil( #Aux_ET00 )
   END_RUNG
   // the same network as SCL:
   #Aux_ET00 := #Aux_ET00 AND NOT #Mx_ET10 AND NOT #Mx_ET10Doble AND NOT #Mx_ET11 AND NOT #Mx_ET12 AND NOT #Mx_ET110 AND NOT #Mx_ET111;
END_REGION

REGION Network 27: ---
   RUNG wire#powerrail
      Contact( #Aux_ET00 )
      I_Contact( #Mx_ET00 )
      I_Contact( #Mx_ET01 )
      I_Contact( #Mx_ET02 )
      I_Contact( #Mx_ET06 )
      I_Contact( #Mx_ET07 )
      I_Contact( #Mx_ET08 )
      I_Contact( #Mx_ET09 )
      S_SR(operand := #Mx_ET00, r1 := wire#w1)
   END_RUNG
   RUNG wire#powerrail
      Contact( #Mx_ET01 )
   END_RUNG wire#w1
   RUNG wire#powerrail
      Contact( #Mx_ET06 )
   END_RUNG wire#w1
   // the same network as SCL:
   IF #Aux_ET00 AND NOT #Mx_ET00 AND NOT #Mx_ET01 AND NOT #Mx_ET02 AND NOT #Mx_ET06 AND NOT #Mx_ET07 AND NOT #Mx_ET08 AND NOT #Mx_ET09 THEN
       #Mx_ET00 := TRUE;   // SR flip-flop
   END_IF;
   IF #Mx_ET01 OR #Mx_ET06 THEN #Mx_ET00 := FALSE; END_IF;
END_REGION

REGION Network 28: TMP - Espera En Tension
   RUNG wire#powerrail
      #TMP_EnTension(R := wire#w1, IN := #EnTension, PV := "V_TMP_EsperaEnTension", BaseUnidades_ms := "CTE_BaseUnidades_1ms", QU =>, QD =>, CVU =>, CVD =>)
   END_RUNG
   RUNG wire#powerrail
      I_Contact( #EnTension )
   END_RUNG wire#w1
   // the same network as SCL:
   #TMP_EnTension(IN := #EnTension,   // "FB910_CNT_UHS"
                  R := NOT #EnTension,
                  PV := "V_TMP_EsperaEnTension",
                  BaseUnidades_ms := "CTE_BaseUnidades_1ms");
END_REGION

REGION Network 29: ERROR - Termico
   RUNG wire#powerrail
      Contact( #EstadoZona.Rearme_CBx )
      S_RS(operand := #EstadoVI.Err_Termico_E1_E3, s1 := wire#w1)
      S_Coil( #EstadoVI.Error_Mx )
   END_RUNG
   RUNG wire#powerrail
      I_Contact( #Termico_Tx )
      Contact( #TMP_EnTension.QU )
   END_RUNG wire#w1
   // the same network as SCL:
   IF #EstadoZona.Rearme_CBx THEN
       #EstadoVI.Err_Termico_E1_E3 := FALSE;   // RS flip-flop
   END_IF;
   IF NOT #Termico_Tx AND #TMP_EnTension.QU THEN #EstadoVI.Err_Termico_E1_E3 := TRUE; END_IF;
   IF #EstadoVI.Err_Termico_E1_E3 THEN #EstadoVI.Error_Mx := TRUE; END_IF;
END_REGION

REGION Network 30: ERROR - Mesa Ocupada
   RUNG wire#powerrail
      Contact( #EstadoZona.Rearme_CBx )
      S_RS(operand := #EstadoVI.Err_Mesa_Ocupada, s1 := wire#w2)
      S_Coil( #EstadoVI.Error_Mx )
   END_RUNG
   RUNG wire#powerrail
      Contact( #Mx_ET01 )
      Contact( #AVTF_MAnt_Mx )
      wire#w1
      Contact( #pHsMx_1 )
   END_RUNG wire#w2
   RUNG wire#w1
      Contact( #pHsMx_2 )
   END_RUNG wire#w2
   // the same network as SCL:
   IF #EstadoZona.Rearme_CBx THEN
       #EstadoVI.Err_Mesa_Ocupada := FALSE;   // RS flip-flop
   END_IF;
   IF #Mx_ET01 AND #AVTF_MAnt_Mx AND (#pHsMx_1 OR #pHsMx_2) THEN #EstadoVI.Err_Mesa_Ocupada := TRUE; END_IF;
   IF #EstadoVI.Err_Mesa_Ocupada THEN #EstadoVI.Error_Mx := TRUE; END_IF;
END_REGION

REGION Network 31: CNT - ERROR - Arrastre
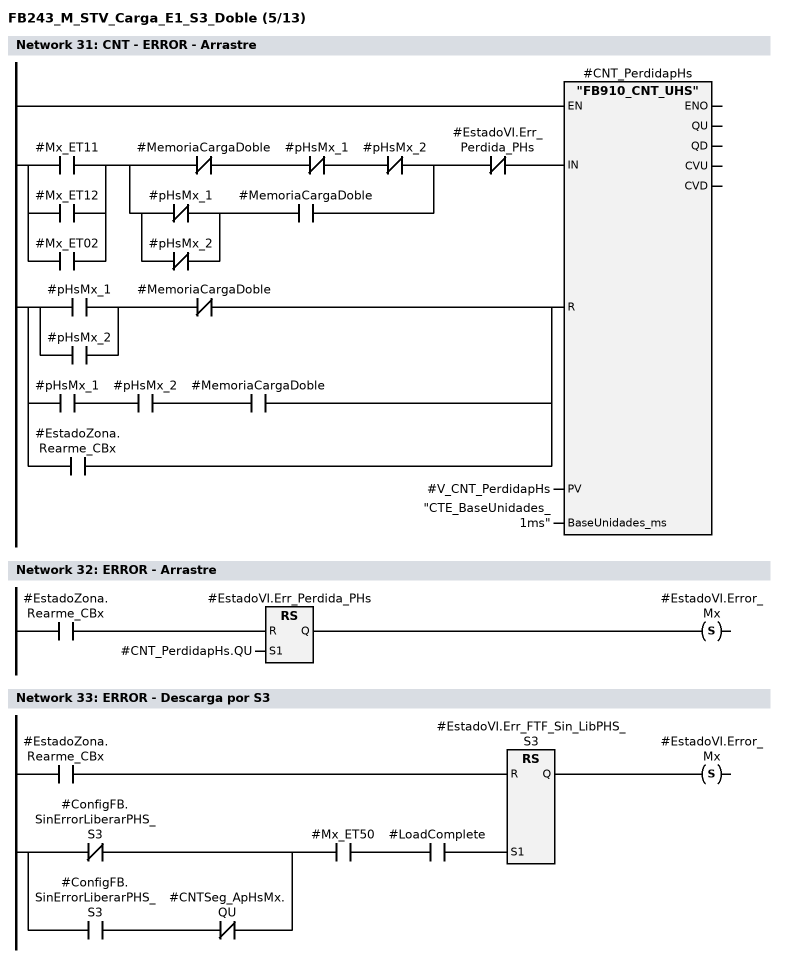
   RUNG wire#powerrail
      #CNT_PerdidapHs(IN := wire#w4, R := wire#w6, PV := #V_CNT_PerdidapHs, BaseUnidades_ms := "CTE_BaseUnidades_1ms", QU =>, QD =>, CVU =>, CVD =>)
   END_RUNG
   RUNG wire#powerrail
      Contact( #Mx_ET11 )
      wire#w1
      I_Contact( #MemoriaCargaDoble )
      I_Contact( #pHsMx_1 )
      I_Contact( #pHsMx_2 )
      wire#w2
      I_Contact( #EstadoVI.Err_Perdida_PHs )
   END_RUNG wire#w4
   RUNG wire#powerrail
      Contact( #Mx_ET12 )
   END_RUNG wire#w1
   RUNG wire#powerrail
      Contact( #Mx_ET02 )
   END_RUNG wire#w1
   RUNG wire#w1
      I_Contact( #pHsMx_1 )
      wire#w3
      Contact( #MemoriaCargaDoble )
   END_RUNG wire#w2
   RUNG wire#w1
      I_Contact( #pHsMx_2 )
   END_RUNG wire#w3
   RUNG wire#powerrail
      Contact( #pHsMx_1 )
      wire#w5
      I_Contact( #MemoriaCargaDoble )
   END_RUNG wire#w6
   RUNG wire#powerrail
      Contact( #pHsMx_2 )
   END_RUNG wire#w5
   RUNG wire#powerrail
      Contact( #pHsMx_1 )
      Contact( #pHsMx_2 )
      Contact( #MemoriaCargaDoble )
   END_RUNG wire#w6
   RUNG wire#powerrail
      Contact( #EstadoZona.Rearme_CBx )
   END_RUNG wire#w6
   // the same network as SCL:
   #CNT_PerdidapHs(IN := (#Mx_ET11 OR #Mx_ET12 OR #Mx_ET02) AND ((NOT #MemoriaCargaDoble AND NOT #pHsMx_1 AND NOT #pHsMx_2) OR ((NOT #pHsMx_1 OR NOT #pHsMx_2) AND #MemoriaCargaDoble)) AND NOT #EstadoVI.Err_Perdida_PHs,   // "FB910_CNT_UHS"
                   R := ((#pHsMx_1 OR #pHsMx_2) AND NOT #MemoriaCargaDoble) OR (#pHsMx_1 AND #pHsMx_2 AND #MemoriaCargaDoble) OR #EstadoZona.Rearme_CBx,
                   PV := #V_CNT_PerdidapHs,
                   BaseUnidades_ms := "CTE_BaseUnidades_1ms");
END_REGION

REGION Network 32: ERROR - Arrastre
   RUNG wire#powerrail
      Contact( #EstadoZona.Rearme_CBx )
      S_RS(operand := #EstadoVI.Err_Perdida_PHs, s1 := #CNT_PerdidapHs.QU)
      S_Coil( #EstadoVI.Error_Mx )
   END_RUNG
   // the same network as SCL:
   IF #EstadoZona.Rearme_CBx THEN
       #EstadoVI.Err_Perdida_PHs := FALSE;   // RS flip-flop
   END_IF;
   IF #CNT_PerdidapHs.QU THEN #EstadoVI.Err_Perdida_PHs := TRUE; END_IF;
   IF #EstadoVI.Err_Perdida_PHs THEN #EstadoVI.Error_Mx := TRUE; END_IF;
END_REGION

REGION Network 33: ERROR - Descarga por S3
   RUNG wire#powerrail
      Contact( #EstadoZona.Rearme_CBx )
      S_RS(operand := #EstadoVI.Err_FTF_Sin_LibPHS_S3, s1 := wire#w2)
      S_Coil( #EstadoVI.Error_Mx )
   END_RUNG
   RUNG wire#powerrail
      I_Contact( #ConfigFB.SinErrorLiberarPHS_S3 )
      wire#w1
      Contact( #Mx_ET50 )
      Contact( #LoadComplete )
   END_RUNG wire#w2
   RUNG wire#powerrail
      Contact( #ConfigFB.SinErrorLiberarPHS_S3 )
      I_Contact( #CNTSeg_ApHsMx.QU )
   END_RUNG wire#w1
   // the same network as SCL:
   IF #EstadoZona.Rearme_CBx THEN
       #EstadoVI.Err_FTF_Sin_LibPHS_S3 := FALSE;   // RS flip-flop
   END_IF;
   IF (NOT #ConfigFB.SinErrorLiberarPHS_S3 OR (#ConfigFB.SinErrorLiberarPHS_S3 AND NOT #CNTSeg_ApHsMx.QU)) AND #Mx_ET50 AND #LoadComplete THEN
       #EstadoVI.Err_FTF_Sin_LibPHS_S3 := TRUE;
   END_IF;
   IF #EstadoVI.Err_FTF_Sin_LibPHS_S3 THEN #EstadoVI.Error_Mx := TRUE; END_IF;
END_REGION

REGION Network 34: TMP - ERROR - TimeOut Avance
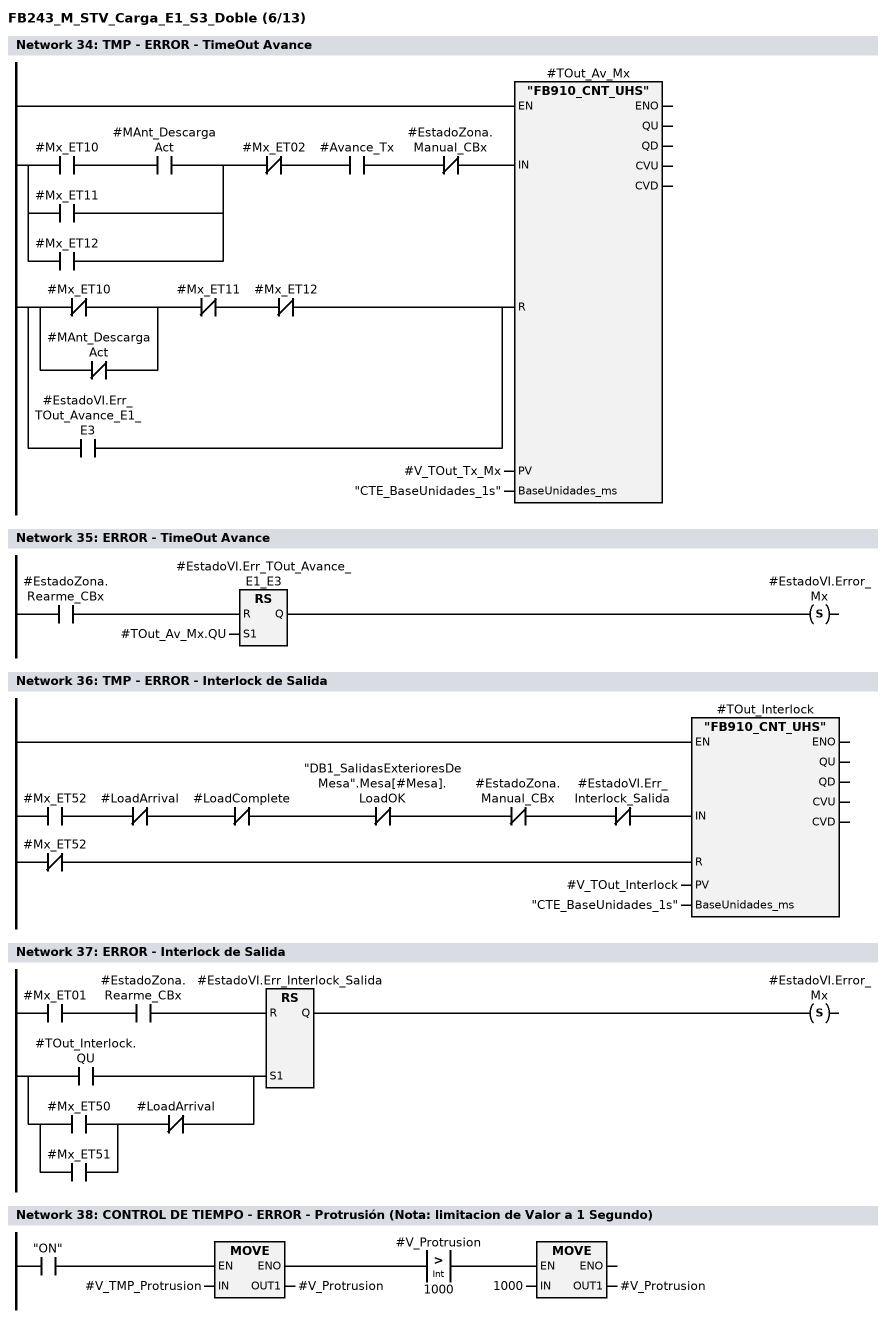
   RUNG wire#powerrail
      #TOut_Av_Mx(IN := wire#w2, R := wire#w4, PV := #V_TOut_Tx_Mx, BaseUnidades_ms := "CTE_BaseUnidades_1s", QU =>, QD =>, CVU =>, CVD =>)
   END_RUNG
   RUNG wire#powerrail
      Contact( #Mx_ET10 )
      Contact( #MAnt_DescargaAct )
      wire#w1
      I_Contact( #Mx_ET02 )
      Contact( #Avance_Tx )
      I_Contact( #EstadoZona.Manual_CBx )
   END_RUNG wire#w2
   RUNG wire#powerrail
      Contact( #Mx_ET11 )
   END_RUNG wire#w1
   RUNG wire#powerrail
      Contact( #Mx_ET12 )
   END_RUNG wire#w1
   RUNG wire#powerrail
      I_Contact( #Mx_ET10 )
      wire#w3
      I_Contact( #Mx_ET11 )
      I_Contact( #Mx_ET12 )
   END_RUNG wire#w4
   RUNG wire#powerrail
      I_Contact( #MAnt_DescargaAct )
   END_RUNG wire#w3
   RUNG wire#powerrail
      Contact( #EstadoVI.Err_TOut_Avance_E1_E3 )
   END_RUNG wire#w4
   // the same network as SCL:
   #TOut_Av_Mx(IN := ((#Mx_ET10 AND #MAnt_DescargaAct) OR #Mx_ET11 OR #Mx_ET12) AND NOT #Mx_ET02 AND #Avance_Tx AND NOT #EstadoZona.Manual_CBx,   // "FB910_CNT_UHS"
               R := ((NOT #Mx_ET10 OR NOT #MAnt_DescargaAct) AND NOT #Mx_ET11 AND NOT #Mx_ET12) OR #EstadoVI.Err_TOut_Avance_E1_E3,
               PV := #V_TOut_Tx_Mx,
               BaseUnidades_ms := "CTE_BaseUnidades_1s");
END_REGION

REGION Network 35: ERROR - TimeOut Avance
   RUNG wire#powerrail
      Contact( #EstadoZona.Rearme_CBx )
      S_RS(operand := #EstadoVI.Err_TOut_Avance_E1_E3, s1 := #TOut_Av_Mx.QU)
      S_Coil( #EstadoVI.Error_Mx )
   END_RUNG
   // the same network as SCL:
   IF #EstadoZona.Rearme_CBx THEN
       #EstadoVI.Err_TOut_Avance_E1_E3 := FALSE;   // RS flip-flop
   END_IF;
   IF #TOut_Av_Mx.QU THEN #EstadoVI.Err_TOut_Avance_E1_E3 := TRUE; END_IF;
   IF #EstadoVI.Err_TOut_Avance_E1_E3 THEN #EstadoVI.Error_Mx := TRUE; END_IF;
END_REGION

REGION Network 36: TMP - ERROR - Interlock de Salida
   RUNG wire#powerrail
      #TOut_Interlock(IN := wire#w1, R := wire#w2, PV := #V_TOut_Interlock, BaseUnidades_ms := "CTE_BaseUnidades_1s", QU =>, QD =>, CVU =>, CVD =>)
   END_RUNG
   RUNG wire#powerrail
      Contact( #Mx_ET52 )
      I_Contact( #LoadArrival )
      I_Contact( #LoadComplete )
      I_Contact( "DB1_SalidasExterioresDeMesa".Mesa[#Mesa].LoadOK )
      I_Contact( #EstadoZona.Manual_CBx )
      I_Contact( #EstadoVI.Err_Interlock_Salida )
   END_RUNG wire#w1
   RUNG wire#powerrail
      I_Contact( #Mx_ET52 )
   END_RUNG wire#w2
   // the same network as SCL:
   #TOut_Interlock(IN := #Mx_ET52 AND NOT #LoadArrival AND NOT #LoadComplete AND NOT "DB1_SalidasExterioresDeMesa".Mesa[#Mesa].LoadOK AND NOT #EstadoZona.Manual_CBx AND NOT #EstadoVI.Err_Interlock_Salida,   // "FB910_CNT_UHS"
                   R := NOT #Mx_ET52,
                   PV := #V_TOut_Interlock,
                   BaseUnidades_ms := "CTE_BaseUnidades_1s");
END_REGION

REGION Network 37: ERROR - Interlock de Salida
   RUNG wire#powerrail
      Contact( #Mx_ET01 )
      Contact( #EstadoZona.Rearme_CBx )
      S_RS(operand := #EstadoVI.Err_Interlock_Salida, s1 := wire#w2)
      S_Coil( #EstadoVI.Error_Mx )
   END_RUNG
   RUNG wire#powerrail
      Contact( #TOut_Interlock.QU )
   END_RUNG wire#w2
   RUNG wire#powerrail
      Contact( #Mx_ET50 )
      wire#w1
      I_Contact( #LoadArrival )
   END_RUNG wire#w2
   RUNG wire#powerrail
      Contact( #Mx_ET51 )
   END_RUNG wire#w1
   // the same network as SCL:
   IF #Mx_ET01 AND #EstadoZona.Rearme_CBx THEN
       #EstadoVI.Err_Interlock_Salida := FALSE;   // RS flip-flop
   END_IF;
   IF #TOut_Interlock.QU OR ((#Mx_ET50 OR #Mx_ET51) AND NOT #LoadArrival) THEN
       #EstadoVI.Err_Interlock_Salida := TRUE;
   END_IF;
   IF #EstadoVI.Err_Interlock_Salida THEN #EstadoVI.Error_Mx := TRUE; END_IF;
END_REGION

REGION Network 38: CONTROL DE TIEMPO - ERROR - Protrusión (Nota: limitacion de Valor a 1 Segundo)
   RUNG wire#powerrail
      Contact( "ON" )
      Move(in := #V_TMP_Protrusion, out1 => #V_Protrusion)
      { S7_Templates := "SrcType := Int" } GT_Contact(in1 := #V_Protrusion, in2 := 1000)
      Move(in := 1000, out1 => #V_Protrusion)
   END_RUNG
   // the same network as SCL:
   IF "ON" THEN #V_Protrusion := #V_TMP_Protrusion; END_IF;
   IF "ON" AND (#V_Protrusion > 1000) THEN #V_Protrusion := 1000; END_IF;
END_REGION

REGION Network 39: TMP - ERROR - Protrusión
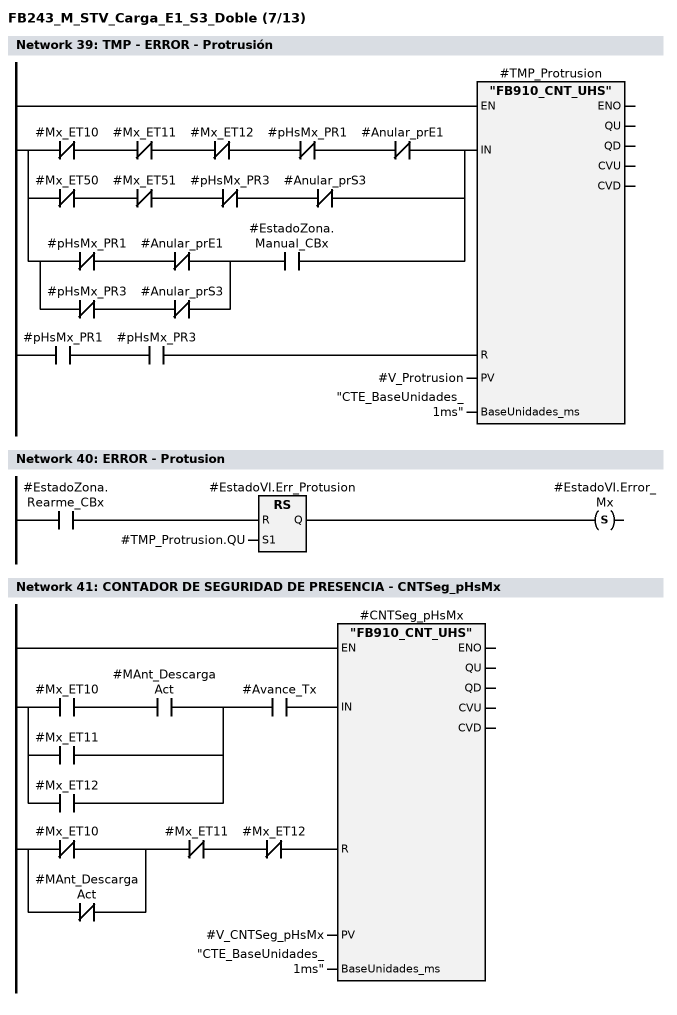
   RUNG wire#powerrail
      #TMP_Protrusion(IN := wire#w2, R := wire#w3, PV := #V_Protrusion, BaseUnidades_ms := "CTE_BaseUnidades_1ms", QU =>, QD =>, CVU =>, CVD =>)
   END_RUNG
   RUNG wire#powerrail
      I_Contact( #Mx_ET10 )
      I_Contact( #Mx_ET11 )
      I_Contact( #Mx_ET12 )
      I_Contact( #pHsMx_PR1 )
      I_Contact( #Anular_prE1 )
   END_RUNG wire#w2
   RUNG wire#powerrail
      I_Contact( #Mx_ET50 )
      I_Contact( #Mx_ET51 )
      I_Contact( #pHsMx_PR3 )
      I_Contact( #Anular_prS3 )
   END_RUNG wire#w2
   RUNG wire#powerrail
      I_Contact( #pHsMx_PR1 )
      I_Contact( #Anular_prE1 )
      wire#w1
      Contact( #EstadoZona.Manual_CBx )
   END_RUNG wire#w2
   RUNG wire#powerrail
      I_Contact( #pHsMx_PR3 )
      I_Contact( #Anular_prS3 )
   END_RUNG wire#w1
   RUNG wire#powerrail
      Contact( #pHsMx_PR1 )
      Contact( #pHsMx_PR3 )
   END_RUNG wire#w3
   // the same network as SCL:
   #TMP_Protrusion(IN := (NOT #Mx_ET10 AND NOT #Mx_ET11 AND NOT #Mx_ET12 AND NOT #pHsMx_PR1 AND NOT #Anular_prE1) OR (NOT #Mx_ET50 AND NOT #Mx_ET51 AND NOT #pHsMx_PR3 AND NOT #Anular_prS3) OR (((NOT #pHsMx_PR1 AND NOT #Anular_prE1) OR (NOT #pHsMx_PR3 AND NOT #Anular_prS3)) AND #EstadoZona.Manual_CBx),   // "FB910_CNT_UHS"
                   R := #pHsMx_PR1 AND #pHsMx_PR3,
                   PV := #V_Protrusion,
                   BaseUnidades_ms := "CTE_BaseUnidades_1ms");
END_REGION

REGION Network 40: ERROR - Protusion
   RUNG wire#powerrail
      Contact( #EstadoZona.Rearme_CBx )
      S_RS(operand := #EstadoVI.Err_Protusion, s1 := #TMP_Protrusion.QU)
      S_Coil( #EstadoVI.Error_Mx )
   END_RUNG
   // the same network as SCL:
   IF #EstadoZona.Rearme_CBx THEN
       #EstadoVI.Err_Protusion := FALSE;   // RS flip-flop
   END_IF;
   IF #TMP_Protrusion.QU THEN #EstadoVI.Err_Protusion := TRUE; END_IF;
   IF #EstadoVI.Err_Protusion THEN #EstadoVI.Error_Mx := TRUE; END_IF;
END_REGION

REGION Network 41: CONTADOR DE SEGURIDAD DE PRESENCIA - CNTSeg_pHsMx
   RUNG wire#powerrail
      #CNTSeg_pHsMx(IN := wire#w2, R := wire#w4, PV := #V_CNTSeg_pHsMx, BaseUnidades_ms := "CTE_BaseUnidades_1ms", QU =>, QD =>, CVU =>, CVD =>)
   END_RUNG
   RUNG wire#powerrail
      Contact( #Mx_ET10 )
      Contact( #MAnt_DescargaAct )
      wire#w1
      Contact( #Avance_Tx )
   END_RUNG wire#w2
   RUNG wire#powerrail
      Contact( #Mx_ET11 )
   END_RUNG wire#w1
   RUNG wire#powerrail
      Contact( #Mx_ET12 )
   END_RUNG wire#w1
   RUNG wire#powerrail
      I_Contact( #Mx_ET10 )
      wire#w3
      I_Contact( #Mx_ET11 )
      I_Contact( #Mx_ET12 )
   END_RUNG wire#w4
   RUNG wire#powerrail
      I_Contact( #MAnt_DescargaAct )
   END_RUNG wire#w3
   // the same network as SCL:
   #CNTSeg_pHsMx(IN := ((#Mx_ET10 AND #MAnt_DescargaAct) OR #Mx_ET11 OR #Mx_ET12) AND #Avance_Tx,   // "FB910_CNT_UHS"
                 R := (NOT #Mx_ET10 OR NOT #MAnt_DescargaAct) AND NOT #Mx_ET11 AND NOT #Mx_ET12,
                 PV := #V_CNTSeg_pHsMx,
                 BaseUnidades_ms := "CTE_BaseUnidades_1ms");
END_REGION

REGION Network 42: CONTADOR DE PRESENCIA - CNT_pHsMx
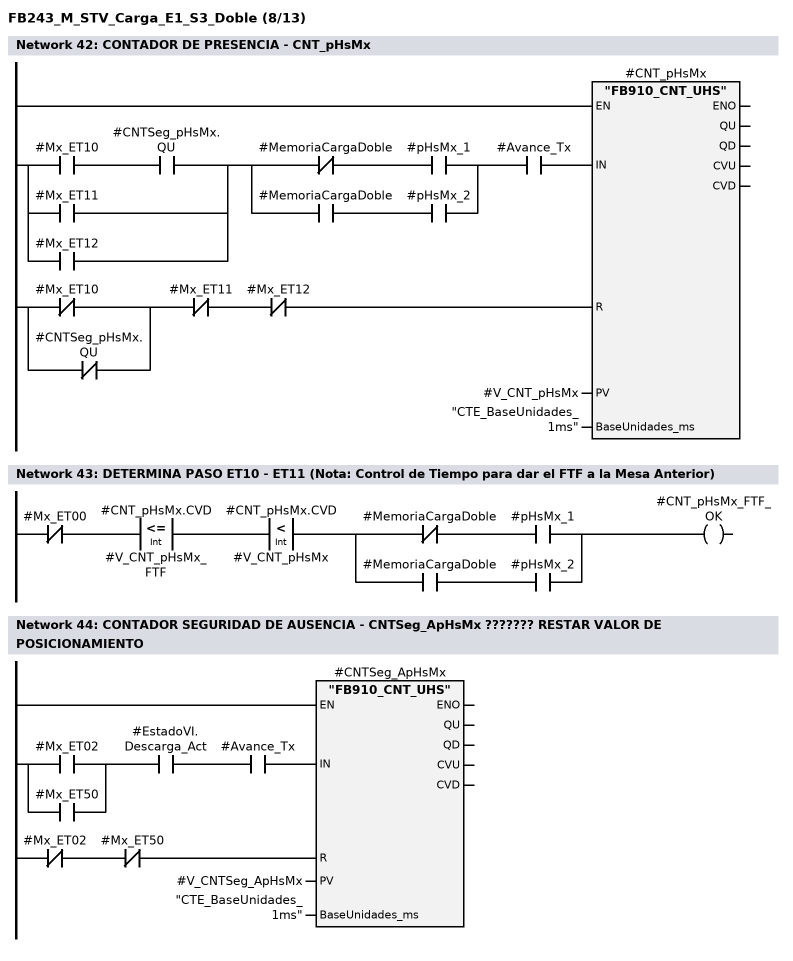
   RUNG wire#powerrail
      #CNT_pHsMx(IN := wire#w3, R := wire#w5, PV := #V_CNT_pHsMx, BaseUnidades_ms := "CTE_BaseUnidades_1ms", QU =>, QD =>, CVU =>, CVD =>)
   END_RUNG
   RUNG wire#powerrail
      Contact( #Mx_ET10 )
      Contact( #CNTSeg_pHsMx.QU )
      wire#w1
      I_Contact( #MemoriaCargaDoble )
      Contact( #pHsMx_1 )
      wire#w2
      Contact( #Avance_Tx )
   END_RUNG wire#w3
   RUNG wire#powerrail
      Contact( #Mx_ET11 )
   END_RUNG wire#w1
   RUNG wire#powerrail
      Contact( #Mx_ET12 )
   END_RUNG wire#w1
   RUNG wire#w1
      Contact( #MemoriaCargaDoble )
      Contact( #pHsMx_2 )
   END_RUNG wire#w2
   RUNG wire#powerrail
      I_Contact( #Mx_ET10 )
      wire#w4
      I_Contact( #Mx_ET11 )
      I_Contact( #Mx_ET12 )
   END_RUNG wire#w5
   RUNG wire#powerrail
      I_Contact( #CNTSeg_pHsMx.QU )
   END_RUNG wire#w4
   // the same network as SCL:
   #CNT_pHsMx(IN := ((#Mx_ET10 AND #CNTSeg_pHsMx.QU) OR #Mx_ET11 OR #Mx_ET12) AND ((NOT #MemoriaCargaDoble AND #pHsMx_1) OR (#MemoriaCargaDoble AND #pHsMx_2)) AND #Avance_Tx,   // "FB910_CNT_UHS"
              R := (NOT #Mx_ET10 OR NOT #CNTSeg_pHsMx.QU) AND NOT #Mx_ET11 AND NOT #Mx_ET12,
              PV := #V_CNT_pHsMx,
              BaseUnidades_ms := "CTE_BaseUnidades_1ms");
END_REGION

REGION Network 43: DETERMINA PASO ET10 - ET11 (Nota: Control de Tiempo para dar el FTF a la Mesa Anterior)
   RUNG wire#powerrail
      I_Contact( #Mx_ET00 )
      { S7_Templates := "SrcType := Int" } LE_Contact(in1 := #CNT_pHsMx.CVD, in2 := #V_CNT_pHsMx_FTF)
      { S7_Templates := "SrcType := Int" } LT_Contact(in1 := #CNT_pHsMx.CVD, in2 := #V_CNT_pHsMx)
      wire#w1
      I_Contact( #MemoriaCargaDoble )
      Contact( #pHsMx_1 )
      wire#w2
      Coil( #CNT_pHsMx_FTF_OK )
   END_RUNG
   RUNG wire#w1
      Contact( #MemoriaCargaDoble )
      Contact( #pHsMx_2 )
   END_RUNG wire#w2
   // the same network as SCL:
   #CNT_pHsMx_FTF_OK := NOT #Mx_ET00 AND (#CNT_pHsMx.CVD <= #V_CNT_pHsMx_FTF) AND (#CNT_pHsMx.CVD < #V_CNT_pHsMx) AND ((NOT #MemoriaCargaDoble AND #pHsMx_1) OR (#MemoriaCargaDoble AND #pHsMx_2));
END_REGION

REGION Network 44: CONTADOR SEGURIDAD DE AUSENCIA - CNTSeg_ApHsMx ??????? RESTAR VALOR DE POSICIONAMIENTO
   RUNG wire#powerrail
      #CNTSeg_ApHsMx(IN := wire#w2, R := wire#w3, PV := #V_CNTSeg_ApHsMx, BaseUnidades_ms := "CTE_BaseUnidades_1ms", QU =>, QD =>, CVU =>, CVD =>)
   END_RUNG
   RUNG wire#powerrail
      Contact( #Mx_ET02 )
      wire#w1
      Contact( #EstadoVI.Descarga_Act )
      Contact( #Avance_Tx )
   END_RUNG wire#w2
   RUNG wire#powerrail
      Contact( #Mx_ET50 )
   END_RUNG wire#w1
   RUNG wire#powerrail
      I_Contact( #Mx_ET02 )
      I_Contact( #Mx_ET50 )
   END_RUNG wire#w3
   // the same network as SCL:
   #CNTSeg_ApHsMx(IN := (#Mx_ET02 OR #Mx_ET50) AND #EstadoVI.Descarga_Act AND #Avance_Tx,   // "FB910_CNT_UHS"
                  R := NOT #Mx_ET02 AND NOT #Mx_ET50,
                  PV := #V_CNTSeg_ApHsMx,
                  BaseUnidades_ms := "CTE_BaseUnidades_1ms");
END_REGION

REGION Network 45: CONTADOR DE LA AUSENCIA - CNT_ApHsMX
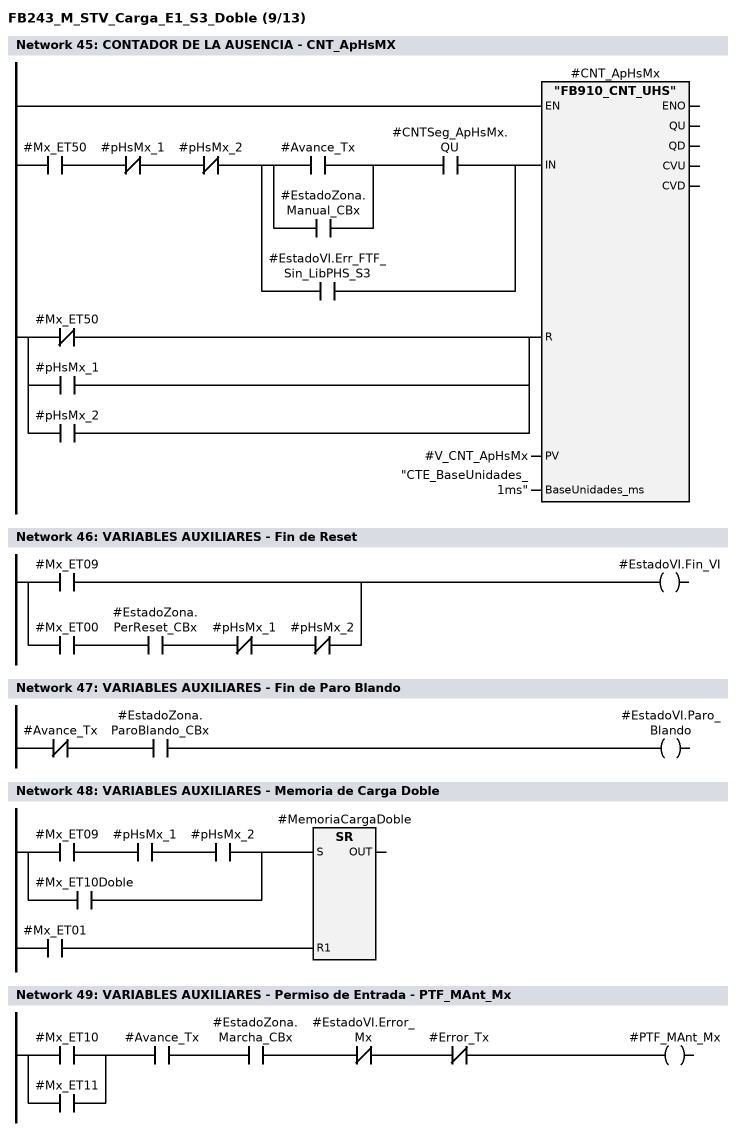
   RUNG wire#powerrail
      #CNT_ApHsMx(IN := wire#w3, R := wire#w4, PV := #V_CNT_ApHsMx, BaseUnidades_ms := "CTE_BaseUnidades_1ms", QU =>, QD =>, CVU =>, CVD =>)
   END_RUNG
   RUNG wire#powerrail
      Contact( #Mx_ET50 )
      I_Contact( #pHsMx_1 )
      I_Contact( #pHsMx_2 )
      wire#w1
      Contact( #Avance_Tx )
      wire#w2
      Contact( #CNTSeg_ApHsMx.QU )
   END_RUNG wire#w3
   RUNG wire#w1
      Contact( #EstadoZona.Manual_CBx )
   END_RUNG wire#w2
   RUNG wire#w1
      Contact( #EstadoVI.Err_FTF_Sin_LibPHS_S3 )
   END_RUNG wire#w3
   RUNG wire#powerrail
      I_Contact( #Mx_ET50 )
   END_RUNG wire#w4
   RUNG wire#powerrail
      Contact( #pHsMx_1 )
   END_RUNG wire#w4
   RUNG wire#powerrail
      Contact( #pHsMx_2 )
   END_RUNG wire#w4
   // the same network as SCL:
   #CNT_ApHsMx(IN := #Mx_ET50 AND NOT #pHsMx_1 AND NOT #pHsMx_2 AND (((#Avance_Tx OR #EstadoZona.Manual_CBx) AND #CNTSeg_ApHsMx.QU) OR #EstadoVI.Err_FTF_Sin_LibPHS_S3),   // "FB910_CNT_UHS"
               R := NOT #Mx_ET50 OR #pHsMx_1 OR #pHsMx_2,
               PV := #V_CNT_ApHsMx,
               BaseUnidades_ms := "CTE_BaseUnidades_1ms");
END_REGION

REGION Network 46: VARIABLES AUXILIARES - Fin de Reset
   RUNG wire#powerrail
      Contact( #Mx_ET09 )
      wire#w1
      Coil( #EstadoVI.Fin_VI )
   END_RUNG
   RUNG wire#powerrail
      Contact( #Mx_ET00 )
      Contact( #EstadoZona.PerReset_CBx )
      I_Contact( #pHsMx_1 )
      I_Contact( #pHsMx_2 )
   END_RUNG wire#w1
   // the same network as SCL:
   #EstadoVI.Fin_VI := #Mx_ET09 OR (#Mx_ET00 AND #EstadoZona.PerReset_CBx AND NOT #pHsMx_1 AND NOT #pHsMx_2);
END_REGION

REGION Network 47: VARIABLES AUXILIARES - Fin de Paro Blando
   RUNG wire#powerrail
      I_Contact( #Avance_Tx )
      Contact( #EstadoZona.ParoBlando_CBx )
      Coil( #EstadoVI.Paro_Blando )
   END_RUNG
   // the same network as SCL:
   #EstadoVI.Paro_Blando := NOT #Avance_Tx AND #EstadoZona.ParoBlando_CBx;
END_REGION

REGION Network 48: VARIABLES AUXILIARES - Memoria de Carga Doble
   RUNG wire#powerrail
      Contact( #Mx_ET09 )
      Contact( #pHsMx_1 )
      Contact( #pHsMx_2 )
      wire#w1
      S_SR(operand := #MemoriaCargaDoble, r1 := wire#w2)
   END_RUNG
   RUNG wire#powerrail
      Contact( #Mx_ET10Doble )
   END_RUNG wire#w1
   RUNG wire#powerrail
      Contact( #Mx_ET01 )
   END_RUNG wire#w2
   // the same network as SCL:
   IF (#Mx_ET09 AND #pHsMx_1 AND #pHsMx_2) OR #Mx_ET10Doble THEN
       #MemoriaCargaDoble := TRUE;   // SR flip-flop
   END_IF;
   IF #Mx_ET01 THEN #MemoriaCargaDoble := FALSE; END_IF;
END_REGION

REGION Network 49: VARIABLES AUXILIARES - Permiso de Entrada - PTF_MAnt_Mx
   RUNG wire#powerrail
      Contact( #Mx_ET10 )
      wire#w1
      Contact( #Avance_Tx )
      Contact( #EstadoZona.Marcha_CBx )
      I_Contact( #EstadoVI.Error_Mx )
      I_Contact( #Error_Tx )
      Coil( #PTF_MAnt_Mx )
   END_RUNG
   RUNG wire#powerrail
      Contact( #Mx_ET11 )
   END_RUNG wire#w1
   // the same network as SCL:
   #PTF_MAnt_Mx := (#Mx_ET10 OR #Mx_ET11) AND #Avance_Tx AND #EstadoZona.Marcha_CBx AND NOT #EstadoVI.Error_Mx AND NOT #Error_Tx;
END_REGION

REGION Network 50: MENSAJES - PRESENCIA
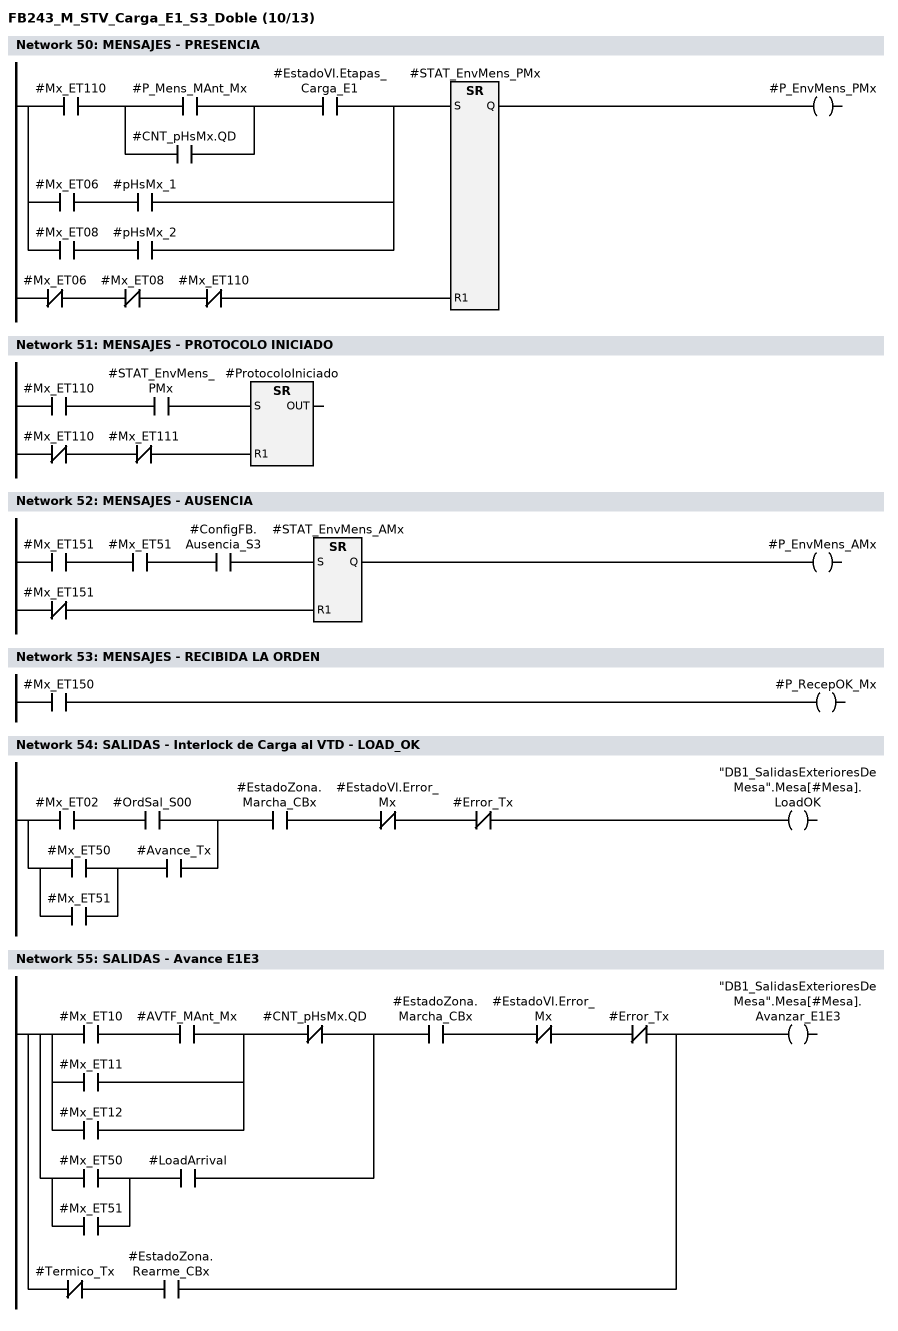
   RUNG wire#powerrail
      Contact( #Mx_ET110 )
      wire#w1
      Contact( #P_Mens_MAnt_Mx )
      wire#w2
      Contact( #EstadoVI.Etapas_Carga_E1 )
      wire#w3
      S_SR(operand := #STAT_EnvMens_PMx, r1 := wire#w4)
      Coil( #P_EnvMens_PMx )
   END_RUNG
   RUNG wire#w1
      Contact( #CNT_pHsMx.QD )
   END_RUNG wire#w2
   RUNG wire#powerrail
      Contact( #Mx_ET06 )
      Contact( #pHsMx_1 )
   END_RUNG wire#w3
   RUNG wire#powerrail
      Contact( #Mx_ET08 )
      Contact( #pHsMx_2 )
   END_RUNG wire#w3
   RUNG wire#powerrail
      I_Contact( #Mx_ET06 )
      I_Contact( #Mx_ET08 )
      I_Contact( #Mx_ET110 )
   END_RUNG wire#w4
   // the same network as SCL:
   IF (#Mx_ET110 AND (#P_Mens_MAnt_Mx OR #CNT_pHsMx.QD) AND #EstadoVI.Etapas_Carga_E1) OR (#Mx_ET06 AND #pHsMx_1) OR (#Mx_ET08 AND #pHsMx_2) THEN
       #STAT_EnvMens_PMx := TRUE;   // SR flip-flop
   END_IF;
   IF NOT #Mx_ET06 AND NOT #Mx_ET08 AND NOT #Mx_ET110 THEN #STAT_EnvMens_PMx := FALSE; END_IF;
   #P_EnvMens_PMx := #STAT_EnvMens_PMx;
END_REGION

REGION Network 51: MENSAJES - PROTOCOLO INICIADO
   RUNG wire#powerrail
      Contact( #Mx_ET110 )
      Contact( #STAT_EnvMens_PMx )
      S_SR(operand := #ProtocoloIniciado, r1 := wire#w1)
   END_RUNG
   RUNG wire#powerrail
      I_Contact( #Mx_ET110 )
      I_Contact( #Mx_ET111 )
   END_RUNG wire#w1
   // the same network as SCL:
   IF #Mx_ET110 AND #STAT_EnvMens_PMx THEN
       #ProtocoloIniciado := TRUE;   // SR flip-flop
   END_IF;
   IF NOT #Mx_ET110 AND NOT #Mx_ET111 THEN #ProtocoloIniciado := FALSE; END_IF;
END_REGION

REGION Network 52: MENSAJES - AUSENCIA
   RUNG wire#powerrail
      Contact( #Mx_ET151 )
      Contact( #Mx_ET51 )
      Contact( #ConfigFB.Ausencia_S3 )
      S_SR(operand := #STAT_EnvMens_AMx, r1 := wire#w1)
      Coil( #P_EnvMens_AMx )
   END_RUNG
   RUNG wire#powerrail
      I_Contact( #Mx_ET151 )
   END_RUNG wire#w1
   // the same network as SCL:
   IF #Mx_ET151 AND #Mx_ET51 AND #ConfigFB.Ausencia_S3 THEN
       #STAT_EnvMens_AMx := TRUE;   // SR flip-flop
   END_IF;
   IF NOT #Mx_ET151 THEN #STAT_EnvMens_AMx := FALSE; END_IF;
   #P_EnvMens_AMx := #STAT_EnvMens_AMx;
END_REGION

REGION Network 53: MENSAJES - RECIBIDA LA ORDEN
   RUNG wire#powerrail
      Contact( #Mx_ET150 )
      Coil( #P_RecepOK_Mx )
   END_RUNG
   // the same network as SCL:
   #P_RecepOK_Mx := #Mx_ET150;
END_REGION

REGION Network 54: SALIDAS - Interlock de Carga al VTD - LOAD_OK
   RUNG wire#powerrail
      Contact( #Mx_ET02 )
      Contact( #OrdSal_S00 )
      wire#w1
      Contact( #EstadoZona.Marcha_CBx )
      I_Contact( #EstadoVI.Error_Mx )
      I_Contact( #Error_Tx )
      Coil( "DB1_SalidasExterioresDeMesa".Mesa[#Mesa].LoadOK )
   END_RUNG
   RUNG wire#powerrail
      Contact( #Mx_ET50 )
      wire#w2
      Contact( #Avance_Tx )
   END_RUNG wire#w1
   RUNG wire#powerrail
      Contact( #Mx_ET51 )
   END_RUNG wire#w2
   // the same network as SCL:
   "DB1_SalidasExterioresDeMesa".Mesa[#Mesa].LoadOK := ((#Mx_ET02 AND #OrdSal_S00) OR ((#Mx_ET50 OR #Mx_ET51) AND #Avance_Tx)) AND #EstadoZona.Marcha_CBx AND NOT #EstadoVI.Error_Mx AND NOT #Error_Tx;
END_REGION

REGION Network 55: SALIDAS - Avance E1E3
   RUNG wire#powerrail
      Contact( #Mx_ET10 )
      Contact( #AVTF_MAnt_Mx )
      wire#w1
      I_Contact( #CNT_pHsMx.QD )
      wire#w2
      Contact( #EstadoZona.Marcha_CBx )
      I_Contact( #EstadoVI.Error_Mx )
      I_Contact( #Error_Tx )
      wire#w4
      Coil( "DB1_SalidasExterioresDeMesa".Mesa[#Mesa].Avanzar_E1E3 )
   END_RUNG
   RUNG wire#powerrail
      Contact( #Mx_ET11 )
   END_RUNG wire#w1
   RUNG wire#powerrail
      Contact( #Mx_ET12 )
   END_RUNG wire#w1
   RUNG wire#powerrail
      Contact( #Mx_ET50 )
      wire#w3
      Contact( #LoadArrival )
   END_RUNG wire#w2
   RUNG wire#powerrail
      Contact( #Mx_ET51 )
   END_RUNG wire#w3
   RUNG wire#powerrail
      I_Contact( #Termico_Tx )
      Contact( #EstadoZona.Rearme_CBx )
   END_RUNG wire#w4
   // the same network as SCL:
   "DB1_SalidasExterioresDeMesa".Mesa[#Mesa].Avanzar_E1E3 := (((((#Mx_ET10 AND #AVTF_MAnt_Mx) OR #Mx_ET11 OR #Mx_ET12) AND NOT #CNT_pHsMx.QD) OR ((#Mx_ET50 OR #Mx_ET51) AND #LoadArrival)) AND #EstadoZona.Marcha_CBx AND NOT #EstadoVI.Error_Mx AND NOT #Error_Tx) OR (NOT #Termico_Tx AND #EstadoZona.Rearme_CBx);
END_REGION

REGION Network 56: SALIDAS - Parar E1E3
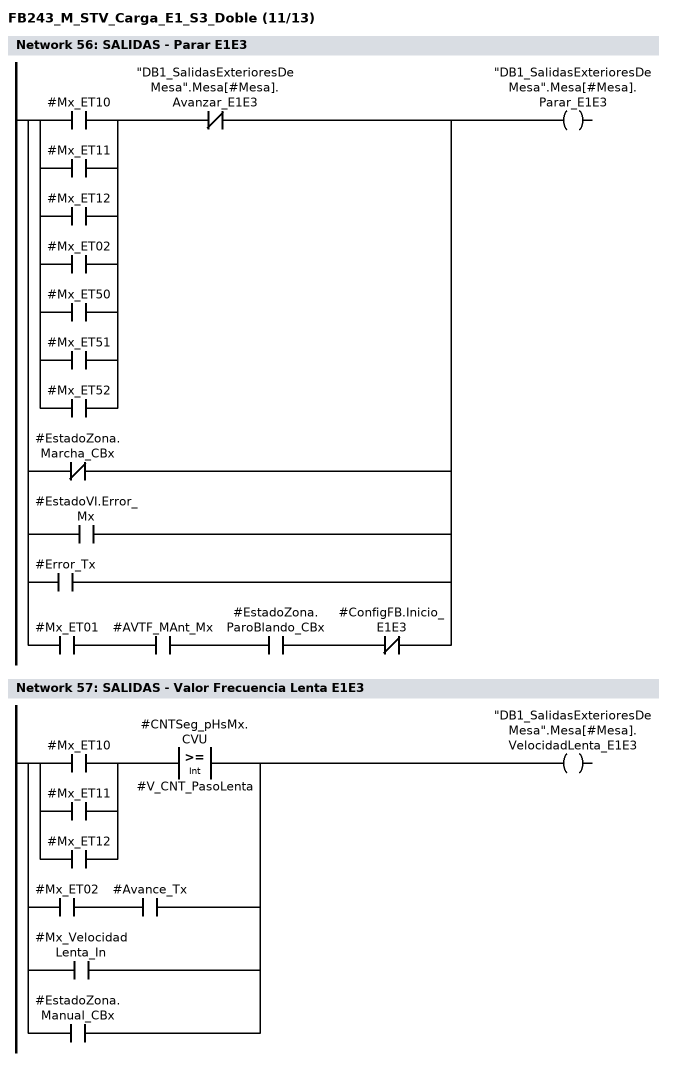
   RUNG wire#powerrail
      Contact( #Mx_ET10 )
      wire#w1
      I_Contact( "DB1_SalidasExterioresDeMesa".Mesa[#Mesa].Avanzar_E1E3 )
      wire#w2
      Coil( "DB1_SalidasExterioresDeMesa".Mesa[#Mesa].Parar_E1E3 )
   END_RUNG
   RUNG wire#powerrail
      Contact( #Mx_ET11 )
   END_RUNG wire#w1
   RUNG wire#powerrail
      Contact( #Mx_ET12 )
   END_RUNG wire#w1
   RUNG wire#powerrail
      Contact( #Mx_ET02 )
   END_RUNG wire#w1
   RUNG wire#powerrail
      Contact( #Mx_ET50 )
   END_RUNG wire#w1
   RUNG wire#powerrail
      Contact( #Mx_ET51 )
   END_RUNG wire#w1
   RUNG wire#powerrail
      Contact( #Mx_ET52 )
   END_RUNG wire#w1
   RUNG wire#powerrail
      I_Contact( #EstadoZona.Marcha_CBx )
   END_RUNG wire#w2
   RUNG wire#powerrail
      Contact( #EstadoVI.Error_Mx )
   END_RUNG wire#w2
   RUNG wire#powerrail
      Contact( #Error_Tx )
   END_RUNG wire#w2
   RUNG wire#powerrail
      Contact( #Mx_ET01 )
      Contact( #AVTF_MAnt_Mx )
      Contact( #EstadoZona.ParoBlando_CBx )
      I_Contact( #ConfigFB.Inicio_E1E3 )
   END_RUNG wire#w2
   // the same network as SCL:
   "DB1_SalidasExterioresDeMesa".Mesa[#Mesa].Parar_E1E3 := ((#Mx_ET10 OR #Mx_ET11 OR #Mx_ET12 OR #Mx_ET02 OR #Mx_ET50 OR #Mx_ET51 OR #Mx_ET52) AND NOT "DB1_SalidasExterioresDeMesa".Mesa[#Mesa].Avanzar_E1E3) OR NOT #EstadoZona.Marcha_CBx OR #EstadoVI.Error_Mx OR #Error_Tx OR (#Mx_ET01 AND #AVTF_MAnt_Mx AND #EstadoZona.ParoBlando_CBx AND NOT #ConfigFB.Inicio_E1E3);
END_REGION

REGION Network 57: SALIDAS - Valor Frecuencia Lenta E1E3
   RUNG wire#powerrail
      Contact( #Mx_ET10 )
      wire#w1
      { S7_Templates := "SrcType := Int" } GE_Contact(in1 := #CNTSeg_pHsMx.CVU, in2 := #V_CNT_PasoLenta)
      wire#w2
      Coil( "DB1_SalidasExterioresDeMesa".Mesa[#Mesa].VelocidadLenta_E1E3 )
   END_RUNG
   RUNG wire#powerrail
      Contact( #Mx_ET11 )
   END_RUNG wire#w1
   RUNG wire#powerrail
      Contact( #Mx_ET12 )
   END_RUNG wire#w1
   RUNG wire#powerrail
      Contact( #Mx_ET02 )
      Contact( #Avance_Tx )
   END_RUNG wire#w2
   RUNG wire#powerrail
      Contact( #Mx_VelocidadLenta_In )
   END_RUNG wire#w2
   RUNG wire#powerrail
      Contact( #EstadoZona.Manual_CBx )
   END_RUNG wire#w2
   // the same network as SCL:
   "DB1_SalidasExterioresDeMesa".Mesa[#Mesa].VelocidadLenta_E1E3 := ((#Mx_ET10 OR #Mx_ET11 OR #Mx_ET12) AND (#CNTSeg_pHsMx.CVU >= #V_CNT_PasoLenta)) OR (#Mx_ET02 AND #Avance_Tx) OR #Mx_VelocidadLenta_In OR #EstadoZona.Manual_CBx;
END_REGION

REGION Network 58: ESTADOS DE LA MESA
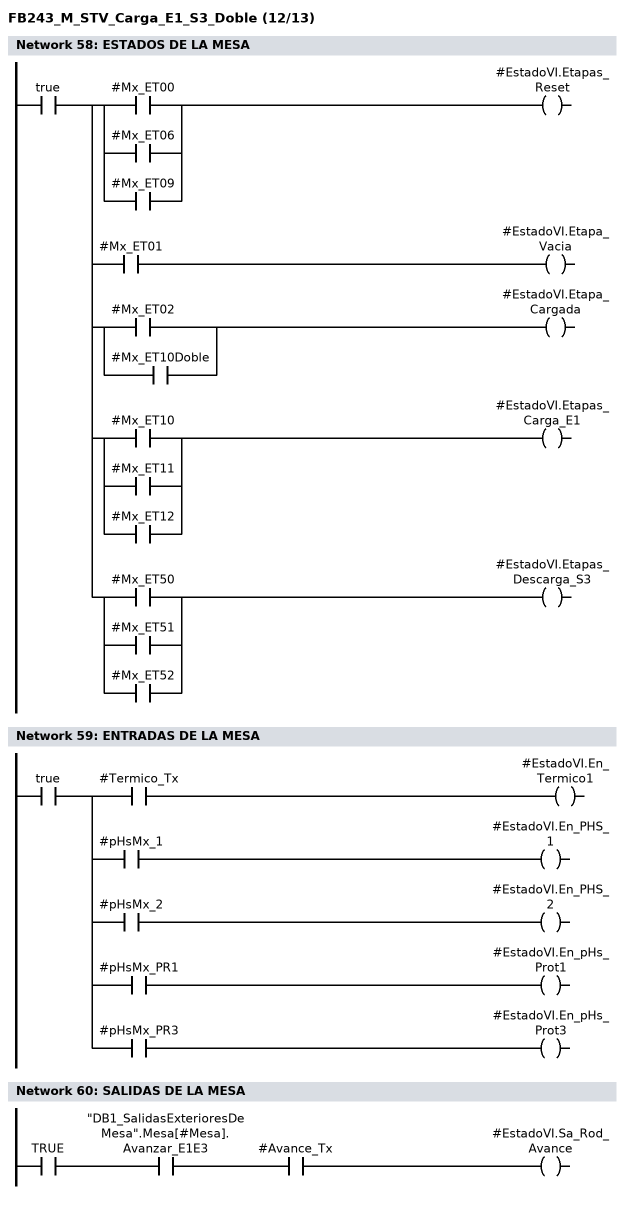
   RUNG wire#powerrail
      Contact( true )
      wire#w1
      Contact( #Mx_ET00 )
      wire#w2
      Coil( #EstadoVI.Etapas_Reset )
   END_RUNG
   RUNG wire#w1
      Contact( #Mx_ET06 )
   END_RUNG wire#w2
   RUNG wire#w1
      Contact( #Mx_ET09 )
   END_RUNG wire#w2
   RUNG wire#w1
      Contact( #Mx_ET01 )
      Coil( #EstadoVI.Etapa_Vacia )
   END_RUNG
   RUNG wire#w1
      Contact( #Mx_ET02 )
      wire#w3
      Coil( #EstadoVI.Etapa_Cargada )
   END_RUNG
   RUNG wire#w1
      Contact( #Mx_ET10Doble )
   END_RUNG wire#w3
   RUNG wire#w1
      Contact( #Mx_ET10 )
      wire#w4
      Coil( #EstadoVI.Etapas_Carga_E1 )
   END_RUNG
   RUNG wire#w1
      Contact( #Mx_ET11 )
   END_RUNG wire#w4
   RUNG wire#w1
      Contact( #Mx_ET12 )
   END_RUNG wire#w4
   RUNG wire#w1
      Contact( #Mx_ET50 )
      wire#w5
      Coil( #EstadoVI.Etapas_Descarga_S3 )
   END_RUNG
   RUNG wire#w1
      Contact( #Mx_ET51 )
   END_RUNG wire#w5
   RUNG wire#w1
      Contact( #Mx_ET52 )
   END_RUNG wire#w5
   // the same network as SCL:
   #EstadoVI.Etapas_Reset := true AND (#Mx_ET00 OR #Mx_ET06 OR #Mx_ET09);
   #EstadoVI.Etapa_Vacia := true AND #Mx_ET01;
   #EstadoVI.Etapa_Cargada := true AND (#Mx_ET02 OR #Mx_ET10Doble);
   #EstadoVI.Etapas_Carga_E1 := true AND (#Mx_ET10 OR #Mx_ET11 OR #Mx_ET12);
   #EstadoVI.Etapas_Descarga_S3 := true AND (#Mx_ET50 OR #Mx_ET51 OR #Mx_ET52);
END_REGION

REGION Network 59: ENTRADAS DE LA MESA
   RUNG wire#powerrail
      Contact( true )
      wire#w1
      Contact( #Termico_Tx )
      Coil( #EstadoVI.En_Termico1 )
   END_RUNG
   RUNG wire#w1
      Contact( #pHsMx_1 )
      Coil( #EstadoVI.En_PHS_1 )
   END_RUNG
   RUNG wire#w1
      Contact( #pHsMx_2 )
      Coil( #EstadoVI.En_PHS_2 )
   END_RUNG
   RUNG wire#w1
      Contact( #pHsMx_PR1 )
      Coil( #EstadoVI.En_pHs_Prot1 )
   END_RUNG
   RUNG wire#w1
      Contact( #pHsMx_PR3 )
      Coil( #EstadoVI.En_pHs_Prot3 )
   END_RUNG
   // the same network as SCL:
   #EstadoVI.En_Termico1 := true AND #Termico_Tx;
   #EstadoVI.En_PHS_1 := true AND #pHsMx_1;
   #EstadoVI.En_PHS_2 := true AND #pHsMx_2;
   #EstadoVI.En_pHs_Prot1 := true AND #pHsMx_PR1;
   #EstadoVI.En_pHs_Prot3 := true AND #pHsMx_PR3;
END_REGION

REGION Network 60: SALIDAS DE LA MESA
   RUNG wire#powerrail
      Contact( TRUE )
      Contact( "DB1_SalidasExterioresDeMesa".Mesa[#Mesa].Avanzar_E1E3 )
      Contact( #Avance_Tx )
      Coil( #EstadoVI.Sa_Rod_Avance )
   END_RUNG
   // the same network as SCL:
   #EstadoVI.Sa_Rod_Avance := TRUE AND "DB1_SalidasExterioresDeMesa".Mesa[#Mesa].Avanzar_E1E3 AND #Avance_Tx;
END_REGION

REGION Network 61: INTERLOCK PARA LA PANTALLA
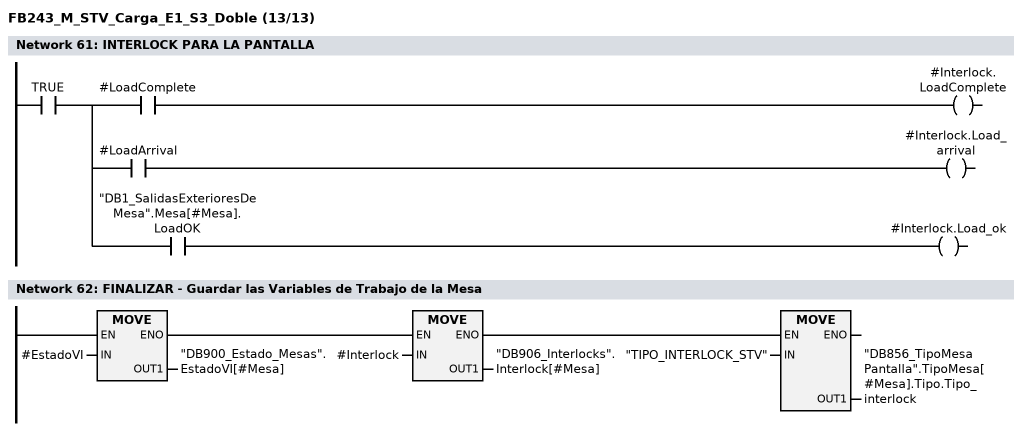
   RUNG wire#powerrail
      Contact( TRUE )
      wire#w1
      Contact( #LoadComplete )
      Coil( #Interlock.LoadComplete )
   END_RUNG
   RUNG wire#w1
      Contact( #LoadArrival )
      Coil( #Interlock.Load_arrival )
   END_RUNG
   RUNG wire#w1
      Contact( "DB1_SalidasExterioresDeMesa".Mesa[#Mesa].LoadOK )
      Coil( #Interlock.Load_ok )
   END_RUNG
   // the same network as SCL:
   #Interlock.LoadComplete := TRUE AND #LoadComplete;
   #Interlock.Load_arrival := TRUE AND #LoadArrival;
   #Interlock.Load_ok := TRUE AND "DB1_SalidasExterioresDeMesa".Mesa[#Mesa].LoadOK;
END_REGION

REGION Network 62: FINALIZAR - Guardar las Variables de Trabajo de la Mesa
   RUNG wire#powerrail
      Move(in := #EstadoVI, out1 => "DB900_Estado_Mesas".EstadoVI[#Mesa])
      Move(in := #Interlock, out1 => "DB906_Interlocks".Interlock[#Mesa])
      Move(in := "TIPO_INTERLOCK_STV", out1 => "DB856_TipoMesaPantalla".TipoMesa[#Mesa].Tipo.Tipo_interlock)
   END_RUNG
   // the same network as SCL:
   "DB900_Estado_Mesas".EstadoVI[#Mesa] := #EstadoVI;
   "DB906_Interlocks".Interlock[#Mesa] := #Interlock;
   "DB856_TipoMesaPantalla".TipoMesa[#Mesa].Tipo.Tipo_interlock := "TIPO_INTERLOCK_STV";
END_REGION
END_FUNCTION_BLOCK
